LIN {X 0,Y 170.6,Z 451.582,A -85,B 0,C 180,E1 -23444.324,E2 -23444.324} C_VEL
LIN {X 0,Y 174.957,Z 460.923,A -85,B 0,C 180,E1 -23446.93,E2 -23446.93} C_VEL
LIN {X 0,Y 177.388,Z 468.584,A -85,B 0,C 180,E1 -23448.831,E2 -23448.831} C_VEL
LIN {X 0,Y 179.037,Z 479.708,A -85,B 0,C 180,E1 -23451.349,E2 -23451.349} C_VEL
LIN {X 0,Y 179.549,Z 490.973,A -85,B 0,C 180,E1 -23454.045,E2 -23454.045} C_VEL
LIN {X 0,Y 179.158,Z 500.868,A -85,B 0,C 180,E1 -23456.688,E2 -23456.688} C_VEL
LIN {X 0,Y 178.388,Z 507.125,A -85,B 0,C 180,E1 -23458.532,E2 -23458.532} C_VEL
LIN {X 0,Y 174.98,Z 515.955,A -85,B 0,C 180,E1 -23461.185,E2 -23461.185} C_VEL
LIN {X 0,Y 171.784,Z 523.786,A -85,B 0,C 180,E1 -23464.166,E2 -23464.166} C_VEL
LIN {X 0,Y 168.834,Z 530.43,A -85,B 0,C 180,E1 -23467.353,E2 -23467.353} C_VEL
LIN {X 0,Y 166.629,Z 535.281,A -85,B 0,C 180,E1 -23470.28,E2 -23470.28} C_VEL
LIN {X 0,Y 164.441,Z 539.995,A -85,B 0,C 180,E1 -23473.871,E2 -23473.871} C_VEL
LIN {X 0,Y 163.057,Z 543.606,A -85,B 0,C 180,E1 -23477.554,E2 -23477.554} C_VEL
LIN {X 0,Y 162.405,Z 545.468,A -85,B 0,C 180,E1 -23480.032,E2 -23480.032} C_VEL
LIN {X 0,Y 162,Z 546.866,A -85,B 0,C 180,E1 -23482.522,E2 -23482.522} C_VEL
LIN {X 0,Y 161.792,Z 547.866,A -85,B 0,C 180,E1 -23485.016,E2 -23485.016} C_VEL
LIN {X 0,Y 161.766,Z 548.53,A -85,B 0,C 180,E1 -23487.776,E2 -23487.776} C_VEL
LIN {X 0,Y 161.899,Z 548.694,A -85,B 0,C 180,E1 -23490,E2 -23490} C_VEL
LIN {X 0,Y 161.765,Z 548.464,A -85,B 0,C 180,E1 -23492.49,E2 -23492.49} C_VEL
LIN {X 0,Y 161.792,Z 547.845,A -85,B 0,C 180,E1 -23494.984,E2 -23494.984} C_VEL
LIN {X 0,Y 162,Z 546.836,A -85,B 0,C 180,E1 -23497.478,E2 -23497.478} C_VEL
LIN {X 0,Y 162.405,Z 545.424,A -85,B 0,C 180,E1 -23499.968,E2 -23499.968} C_VEL
LIN {X 0,Y 163.457,Z 542.468,A -85,B 0,C 180,E1 -23503.679,E2 -23503.679} C_VEL
LIN {X 0,Y 165.07,Z 538.474,A -85,B 0,C 180,E1 -23507.339,E2 -23507.339} C_VEL
LIN {X 0,Y 167.886,Z 532.345,A -85,B 0,C 180,E1 -23511.487,E2 -23511.487} C_VEL
LIN {X 0,Y 170.867,Z 525.858,A -85,B 0,C 180,E1 -23514.829,E2 -23514.829} C_VEL
LIN {X 0,Y 173.339,Z 519.858,A -85,B 0,C 180,E1 -23517.348,E2 -23517.348} C_VEL
LIN {X 0,Y 174.23,Z 516.073,A -85,B 0,C 180,E1 -23518.815,E2 -23518.815} C_VEL
LIN {X 0,Y 174.205,Z 512.249,A -85,B 0,C 180,E1 -23520.33,E2 -23520.33} C_VEL
LIN {X 0,Y 173.132,Z 504.415,A -85,B 0,C 180,E1 -23523.344,E2 -23523.344} C_VEL
LIN {X 0,Y 172.989,Z 498.624,A -85,B 0,C 180,E1 -23525.198,E2 -23525.198} C_VEL
LIN {X 0,Y 173.249,Z 489.2,A -85,B 0,C 180,E1 -23527.785,E2 -23527.785} C_VEL
LIN {X 0,Y 172.79,Z 479.133,A -85,B 0,C 180,E1 -23530.303,E2 -23530.303} C_VEL
LIN {X 0,Y 171.463,Z 470.4,A -85,B 0,C 180,E1 -23532.456,E2 -23532.456} C_VEL
LIN {X 0,Y 169.332,Z 463.748,A -85,B 0,C 180,E1 -23534.279,E2 -23534.279} C_VEL
LIN {X 0,Y 165.519,Z 455.347,A -85,B 0,C 180,E1 -23536.863,E2 -23536.863} C_VEL
LIN {X 0,Y 163.537,Z 451.389,A -85,B 0,C 180,E1 -23538.129,E2 -23538.129} C_VEL
LIN {X 0,Y 161.489,Z 447.46,A -85,B 0,C 180,E1 -23539.426,E2 -23539.426} C_VEL
LIN {X 0,Y 160.888,Z 446.45,A -85,B 0,C 180,E1 -23539.781,E2 -23539.781} C_VEL
LIN {X 0,Y 158.813,Z 443.395,A -85,B 0,C 180,E1 -23540.997,E2 -23540.997} C_VEL
LIN {X 0,Y 158.112,Z 441.187,A -85,B 0,C 180,E1 -23541.578,E2 -23541.578} C_VEL
LIN {X 0,Y 157.962,Z 439.682,A -85,B 0,C 180,E1 -23544.662,E2 -23544.662} C_VEL
LIN {X 0,Y 157.752,Z 438.263,A -85,B 0,C 180,E1 -23547.829,E2 -23547.829} C_VEL
LIN {X 0,Y 157.341,Z 436.003,A -85,B 0,C 180,E1 -23553.47,E2 -23553.47} C_VEL
LIN {X 0,Y 157.395,Z 435.881,A -85,B 0,C 180,E1 -23559.667,E2 -23559.667} C_VEL
LIN {X 0,Y 157.48,Z 435.869,A -85,B 0,C 180,E1 -23564.469,E2 -23564.469} C_VEL
LIN {X 0,Y 157.774,Z 435.833,A -85,B 0,C 180,E1 -23569.736,E2 -23569.736} C_VEL
LIN {X 0,Y 157.826,Z 435.824,A -85,B 0,C 180,E1 -23572.323,E2 -23572.323} C_VEL
LIN {X 0,Y 158.261,Z 435.77,A -85,B 0,C 180,E1 -23580,E2 -23580} C_VEL
LIN {X 0,Y 157.826,Z 435.825,A -85,B 0,C 180,E1 -23587.677,E2 -23587.677} C_VEL
LIN {X 0,Y 157.707,Z 435.839,A -85,B 0,C 180,E1 -23591.363,E2 -23591.363} C_VEL
LIN {X 0,Y 157.48,Z 435.868,A -85,B 0,C 180,E1 -23595.532,E2 -23595.532} C_VEL
LIN {X 0,Y 157.371,Z 435.88,A -85,B 0,C 180,E1 -23600.933,E2 -23600.933} C_VEL
LIN {X 0,Y 157.316,Z 435.888,A -85,B 0,C 180,E1 -23606.685,E2 -23606.685} C_VEL
LIN {X 0,Y 157.279,Z 435.892,A -85,B 0,C 180,E1 -23612.427,E2 -23612.427} C_VEL
LIN {X 0,Y 157.257,Z 435.896,A -85,B 0,C 180,E1 -23617.476,E2 -23617.476} C_VEL
LIN {X 0,Y 157.227,Z 435.906,A -85,B 0,C 180,E1 -23618.11,E2 -23618.11} C_VEL
LIN {X 0,Y 158.173,Z 438.66,A -85,B 0,C 180,E1 -23618.871,E2 -23618.871} C_VEL
LIN {X 0,Y 160.688,Z 441.686,A -85,B 0,C 180,E1 -23620.309,E2 -23620.309} C_VEL
LIN {X 0,Y 162.705,Z 445.357,A -85,B 0,C 180,E1 -23621.615,E2 -23621.615} C_VEL
LIN {X 0,Y 163.922,Z 447.482,A -85,B 0,C 180,E1 -23622.371,E2 -23622.371} C_VEL
LIN {X 0,Y 166.788,Z 452.918,A -85,B 0,C 180,E1 -23624.248,E2 -23624.248} C_VEL
LIN {X 0,Y 170.183,Z 460.491,A -85,B 0,C 180,E1 -23626.703,E2 -23626.703} C_VEL
LIN {X 0,Y 173.03,Z 469.987,A -85,B 0,C 180,E1 -23629.468,E2 -23629.468} C_VEL
LIN {X 0,Y 174.705,Z 480.999,A -85,B 0,C 180,E1 -23632.557,E2 -23632.557} C_VEL
LIN {X 0,Y 175.044,Z 489.187,A -85,B 0,C 180,E1 -23634.944,E2 -23634.944} C_VEL
LIN {X 0,Y 174.851,Z 495.164,A -85,B 0,C 180,E1 -23636.794,E2 -23636.794} C_VEL
LIN {X 0,Y 171.108,Z 504.928,A -85,B 0,C 180,E1 -23639.604,E2 -23639.604} C_VEL
LIN {X 0,Y 167.634,Z 512.925,A -85,B 0,C 180,E1 -23642.537,E2 -23642.537} C_VEL
LIN {X 0,Y 164.104,Z 520.326,A -85,B 0,C 180,E1 -23645.993,E2 -23645.993} C_VEL
LIN {X 0,Y 161.079,Z 526.265,A -85,B 0,C 180,E1 -23649.571,E2 -23649.571} C_VEL
LIN {X 0,Y 158.726,Z 530.952,A -85,B 0,C 180,E1 -23653.274,E2 -23653.274} C_VEL
LIN {X 0,Y 156.932,Z 534.537,A -85,B 0,C 180,E1 -23657.061,E2 -23657.061} C_VEL
LIN {X 0,Y 156.086,Z 536.386,A -85,B 0,C 180,E1 -23659.624,E2 -23659.624} C_VEL
LIN {X 0,Y 155.506,Z 537.773,A -85,B 0,C 180,E1 -23662.208,E2 -23662.208} C_VEL
LIN {X 0,Y 154.905,Z 539.364,A -85,B 0,C 180,E1 -23667.4,E2 -23667.4} C_VEL
LIN {X 0,Y 154.861,Z 539.59,A -85,B 0,C 180,E1 -23670,E2 -23670} C_VEL
LIN {X 0,Y 155.016,Z 539.119,A -85,B 0,C 180,E1 -23674.11,E2 -23674.11} C_VEL
LIN {X 0,Y 155.506,Z 537.842,A -85,B 0,C 180,E1 -23677.793,E2 -23677.793} C_VEL
LIN {X 0,Y 156.086,Z 536.486,A -85,B 0,C 180,E1 -23680.376,E2 -23680.376} C_VEL
LIN {X 0,Y 157.445,Z 533.617,A -85,B 0,C 180,E1 -23684.212,E2 -23684.212} C_VEL
LIN {X 0,Y 159.414,Z 529.724,A -85,B 0,C 180,E1 -23687.976,E2 -23687.976} C_VEL
LIN {X 0,Y 161.939,Z 524.7,A -85,B 0,C 180,E1 -23691.648,E2 -23691.648} C_VEL
LIN {X 0,Y 165.158,Z 518.366,A -85,B 0,C 180,E1 -23695.185,E2 -23695.185} C_VEL
LIN {X 0,Y 168.668,Z 510.778,A -85,B 0,C 180,E1 -23698.48,E2 -23698.48} C_VEL
LIN {X 0,Y 172.046,Z 502.551,A -85,B 0,C 180,E1 -23701.32,E2 -23701.32} C_VEL
LIN {X 0,Y 175.038,Z 494.65,A -85,B 0,C 180,E1 -23703.51,E2 -23703.51} C_VEL
LIN {X 0,Y 175.053,Z 485.144,A -85,B 0,C 180,E1 -23706.412,E2 -23706.412} C_VEL
LIN {X 0,Y 174.124,Z 476.029,A -85,B 0,C 180,E1 -23709.032,E2 -23709.032} C_VEL
LIN {X 0,Y 172.706,Z 468.444,A -85,B 0,C 180,E1 -23711.162,E2 -23711.162} C_VEL
LIN {X 0,Y 170.166,Z 460.375,A -85,B 0,C 180,E1 -23713.527,E2 -23713.527} C_VEL
LIN {X 0,Y 165.678,Z 450.421,A -85,B 0,C 180,E1 -23716.743,E2 -23716.743} C_VEL
LIN {X 0,Y 163.427,Z 446.317,A -85,B 0,C 180,E1 -23718.197,E2 -23718.197} C_VEL
LIN {X 0,Y 160.984,Z 442.422,A -85,B 0,C 180,E1 -23719.707,E2 -23719.707} C_VEL
LIN {X 0,Y 160.22,Z 440.995,A -85,B 0,C 180,E1 -23720.199,E2 -23720.199} C_VEL
LIN {X 0,Y 157.993,Z 438.397,A -85,B 0,C 180,E1 -23721.481,E2 -23721.481} C_VEL
LIN {X 0,Y 157.227,Z 435.899,A -85,B 0,C 180,E1 -23722.204,E2 -23722.204} C_VEL
LIN {X 0,Y 157.292,Z 435.889,A -85,B 0,C 180,E1 -23724.489,E2 -23724.489} C_VEL
LIN {X 0,Y 157.296,Z 435.89,A -85,B 0,C 180,E1 -23728.095,E2 -23728.095} C_VEL
LIN {X 0,Y 157.324,Z 435.883,A -85,B 0,C 180,E1 -23733.466,E2 -23733.466} C_VEL
LIN {X 0,Y 157.396,Z 435.878,A -85,B 0,C 180,E1 -23739.667,E2 -23739.667} C_VEL
LIN {X 0,Y 157.481,Z 435.868,A -85,B 0,C 180,E1 -23744.468,E2 -23744.468} C_VEL
LIN {X 0,Y 157.775,Z 435.833,A -85,B 0,C 180,E1 -23749.736,E2 -23749.736} C_VEL
LIN {X 0,Y 157.827,Z 435.826,A -85,B 0,C 180,E1 -23752.323,E2 -23752.323} C_VEL
LIN {X 0,Y 158.261,Z 435.77,A -85,B 0,C 180,E1 -23760,E2 -23760} C_VEL
LIN {X 0,Y 157.827,Z 435.824,A -85,B 0,C 180,E1 -23767.677,E2 -23767.677} C_VEL
LIN {X 0,Y 157.708,Z 435.839,A -85,B 0,C 180,E1 -23771.363,E2 -23771.363} C_VEL
LIN {X 0,Y 157.488,Z 435.866,A -85,B 0,C 180,E1 -23775.531,E2 -23775.531} C_VEL
LIN {X 0,Y 157.373,Z 435.882,A -85,B 0,C 180,E1 -23780.932,E2 -23780.932} C_VEL
LIN {X 0,Y 157.382,Z 436.144,A -85,B 0,C 180,E1 -23786.732,E2 -23786.732} C_VEL
LIN {X 0,Y 157.715,Z 438.408,A -85,B 0,C 180,E1 -23792.326,E2 -23792.326} C_VEL
LIN {X 0,Y 158.04,Z 440.801,A -85,B 0,C 180,E1 -23797.515,E2 -23797.515} C_VEL
LIN {X 0,Y 158.138,Z 441.341,A -85,B 0,C 180,E1 -23798.352,E2 -23798.352} C_VEL
LIN {X 0,Y 159.193,Z 444.167,A -85,B 0,C 180,E1 -23799.109,E2 -23799.109} C_VEL
LIN {X 0,Y 161.514,Z 447.463,A -85,B 0,C 180,E1 -23800.447,E2 -23800.447} C_VEL
LIN {X 0,Y 163.398,Z 451.165,A -85,B 0,C 180,E1 -23801.659,E2 -23801.659} C_VEL
LIN {X 0,Y 164.568,Z 453.304,A -85,B 0,C 180,E1 -23802.373,E2 -23802.373} C_VEL
LIN {X 0,Y 168.071,Z 460.658,A -85,B 0,C 180,E1 -23804.694,E2 -23804.694} C_VEL
LIN {X 0,Y 171.256,Z 469.263,A -85,B 0,C 180,E1 -23807.171,E2 -23807.171} C_VEL
LIN {X 0,Y 172.513,Z 476.304,A -85,B 0,C 180,E1 -23808.911,E2 -23808.911} C_VEL
LIN {X 0,Y 173.303,Z 485.676,A -85,B 0,C 180,E1 -23811.238,E2 -23811.238} C_VEL
LIN {X 0,Y 173.202,Z 496.91,A -85,B 0,C 180,E1 -23814.247,E2 -23814.247} C_VEL
LIN {X 0,Y 172.404,Z 504.943,A -85,B 0,C 180,E1 -23816.61,E2 -23816.61} C_VEL
LIN {X 0,Y 171.672,Z 508.87,A -85,B 0,C 180,E1 -23817.845,E2 -23817.845} C_VEL
LIN {X 0,Y 168.103,Z 517.33,A -85,B 0,C 180,E1 -23820.577,E2 -23820.577} C_VEL
LIN {X 0,Y 164.638,Z 525.326,A -85,B 0,C 180,E1 -23823.901,E2 -23823.901} C_VEL
LIN {X 0,Y 161.257,Z 532.261,A -85,B 0,C 180,E1 -23827.582,E2 -23827.582} C_VEL
LIN {X 0,Y 158.296,Z 538.357,A -85,B 0,C 180,E1 -23831.893,E2 -23831.893} C_VEL
LIN {X 0,Y 156.531,Z 542.326,A -85,B 0,C 180,E1 -23835.703,E2 -23835.703} C_VEL
LIN {X 0,Y 155.406,Z 545.264,A -85,B 0,C 180,E1 -23839.578,E2 -23839.578} C_VEL
LIN {X 0,Y 154.95,Z 546.662,A -85,B 0,C 180,E1 -23842.179,E2 -23842.179} C_VEL
LIN {X 0,Y 154.712,Z 547.662,A -85,B 0,C 180,E1 -23844.787,E2 -23844.787} C_VEL
LIN {X 0,Y 154.684,Z 548.389,A -85,B 0,C 180,E1 -23848.304,E2 -23848.304} C_VEL
LIN {X 0,Y 154.797,Z 548.49,A -85,B 0,C 180,E1 -23850,E2 -23850} C_VEL
LIN {X 0,Y 154.667,Z 548.26,A -85,B 0,C 180,E1 -23852.604,E2 -23852.604} C_VEL
LIN {X 0,Y 154.712,Z 547.64,A -85,B 0,C 180,E1 -23855.212,E2 -23855.212} C_VEL
LIN {X 0,Y 154.95,Z 546.631,A -85,B 0,C 180,E1 -23857.82,E2 -23857.82} C_VEL
LIN {X 0,Y 155.405,Z 545.219,A -85,B 0,C 180,E1 -23860.422,E2 -23860.422} C_VEL
LIN {X 0,Y 156.53,Z 542.262,A -85,B 0,C 180,E1 -23864.296,E2 -23864.296} C_VEL
LIN {X 0,Y 158.295,Z 538.269,A -85,B 0,C 180,E1 -23868.106,E2 -23868.106} C_VEL
LIN {X 0,Y 161.255,Z 532.138,A -85,B 0,C 180,E1 -23872.417,E2 -23872.417} C_VEL
LIN {X 0,Y 164.561,Z 525.263,A -85,B 0,C 180,E1 -23876.062,E2 -23876.062} C_VEL
LIN {X 0,Y 168.101,Z 517.147,A -85,B 0,C 180,E1 -23879.422,E2 -23879.422} C_VEL
LIN {X 0,Y 171.631,Z 508.636,A -85,B 0,C 180,E1 -23882.163,E2 -23882.163} C_VEL
LIN {X 0,Y 172.869,Z 500.383,A -85,B 0,C 180,E1 -23884.692,E2 -23884.692} C_VEL
LIN {X 0,Y 172.989,Z 498.624,A -85,B 0,C 180,E1 -23885.198,E2 -23885.198} C_VEL
LIN {X 0,Y 172.681,Z 494.345,A -85,B 0,C 180,E1 -23886.531,E2 -23886.531} C_VEL
LIN {X 0,Y 171.427,Z 490.35,A -85,B 0,C 180,E1 -23887.944,E2 -23887.944} C_VEL
LIN {X 0,Y 168.002,Z 482.617,A -85,B 0,C 180,E1 -23890.835,E2 -23890.835} C_VEL
LIN {X 0,Y 166.494,Z 476.796,A -85,B 0,C 180,E1 -23892.645,E2 -23892.645} C_VEL
LIN {X 0,Y 165.046,Z 470.124,A -85,B 0,C 180,E1 -23894.532,E2 -23894.532} C_VEL
LIN {X 0,Y 161.383,Z 460.851,A -85,B 0,C 180,E1 -23897.547,E2 -23897.547} C_VEL
LIN {X 0,Y 159.089,Z 456.083,A -85,B 0,C 180,E1 -23899.233,E2 -23899.233} C_VEL
LIN {X 0,Y 156.754,Z 451.512,A -85,B 0,C 180,E1 -23900.914,E2 -23900.914} C_VEL
LIN {X 0,Y 154.664,Z 447.676,A -85,B 0,C 180,E1 -23902.409,E2 -23902.409} C_VEL
LIN {X 0,Y 153.912,Z 446.339,A -85,B 0,C 180,E1 -23902.93,E2 -23902.93} C_VEL
LIN {X 0,Y 151.726,Z 443.154,A -85,B 0,C 180,E1 -23904.416,E2 -23904.416} C_VEL
LIN {X 0,Y 150.944,Z 440.831,A -85,B 0,C 180,E1 -23905.224,E2 -23905.224} C_VEL
LIN {X 0,Y 150.666,Z 439.2,A -85,B 0,C 180,E1 -23909.129,E2 -23909.129} C_VEL
LIN {X 0,Y 150.431,Z 437.884,A -85,B 0,C 180,E1 -23912.581,E2 -23912.581} C_VEL
LIN {X 0,Y 150.266,Z 436.997,A -85,B 0,C 180,E1 -23915.106,E2 -23915.106} C_VEL
LIN {X 0,Y 150.368,Z 436.756,A -85,B 0,C 180,E1 -23920.903,E2 -23920.903} C_VEL
LIN {X 0,Y 150.465,Z 436.742,A -85,B 0,C 180,E1 -23926.494,E2 -23926.494} C_VEL
LIN {X 0,Y 150.69,Z 436.715,A -85,B 0,C 180,E1 -23929.248,E2 -23929.248} C_VEL
LIN {X 0,Y 150.764,Z 436.706,A -85,B 0,C 180,E1 -23931.961,E2 -23931.961} C_VEL
LIN {X 0,Y 151.221,Z 436.647,A -85,B 0,C 180,E1 -23940,E2 -23940} C_VEL
LIN {X 0,Y 150.764,Z 436.704,A -85,B 0,C 180,E1 -23948.039,E2 -23948.039} C_VEL
LIN {X 0,Y 150.636,Z 436.72,A -85,B 0,C 180,E1 -23951.546,E2 -23951.546} C_VEL
LIN {X 0,Y 150.385,Z 436.751,A -85,B 0,C 180,E1 -23956.284,E2 -23956.284} C_VEL
LIN {X 0,Y 150.352,Z 436.753,A -85,B 0,C 180,E1 -23960.793,E2 -23960.793} C_VEL
LIN {X 0,Y 150.245,Z 436.768,A -85,B 0,C 180,E1 -23967.283,E2 -23967.283} C_VEL
LIN {X 0,Y 150.22,Z 436.771,A -85,B 0,C 180,E1 -23972.635,E2 -23972.635} C_VEL
LIN {X 0,Y 150.222,Z 436.885,A -85,B 0,C 180,E1 -23974.661,E2 -23974.661} C_VEL
LIN {X 0,Y 151.09,Z 439.359,A -85,B 0,C 180,E1 -23975.45,E2 -23975.45} C_VEL
LIN {X 0,Y 153.214,Z 441.722,A -85,B 0,C 180,E1 -23976.852,E2 -23976.852} C_VEL
LIN {X 0,Y 153.8,Z 442.446,A -85,B 0,C 180,E1 -23977.238,E2 -23977.238} C_VEL
LIN {X 0,Y 155.53,Z 445.479,A -85,B 0,C 180,E1 -23978.515,E2 -23978.515} C_VEL
LIN {X 0,Y 156.95,Z 447.413,A -85,B 0,C 180,E1 -23979.442,E2 -23979.442} C_VEL
LIN {X 0,Y 160.981,Z 455.021,A -85,B 0,C 180,E1 -23982.416,E2 -23982.416} C_VEL
LIN {X 0,Y 164.913,Z 464.218,A -85,B 0,C 180,E1 -23985.651,E2 -23985.651} C_VEL
LIN {X 0,Y 167.208,Z 472.415,A -85,B 0,C 180,E1 -23988.25,E2 -23988.25} C_VEL
LIN {X 0,Y 168.59,Z 482.499,A -85,B 0,C 180,E1 -23991.296,E2 -23991.296} C_VEL
LIN {X 0,Y 168.823,Z 491.095,A -85,B 0,C 180,E1 -23993.988,E2 -23993.988} C_VEL
LIN {X 0,Y 168.559,Z 496.426,A -85,B 0,C 180,E1 -23995.745,E2 -23995.745} C_VEL
LIN {X 0,Y 164.739,Z 505.744,A -85,B 0,C 180,E1 -23998.565,E2 -23998.565} C_VEL
LIN {X 0,Y 160.736,Z 514.478,A -85,B 0,C 180,E1 -24001.964,E2 -24001.964} C_VEL
LIN {X 0,Y 157.062,Z 521.642,A -85,B 0,C 180,E1 -24005.55,E2 -24005.55} C_VEL
LIN {X 0,Y 154.431,Z 526.471,A -85,B 0,C 180,E1 -24008.65,E2 -24008.65} C_VEL
LIN {X 0,Y 151.949,Z 531.157,A -85,B 0,C 180,E1 -24012.504,E2 -24012.504} C_VEL
LIN {X 0,Y 150.017,Z 534.742,A -85,B 0,C 180,E1 -24016.453,E2 -24016.453} C_VEL
LIN {X 0,Y 149.111,Z 536.591,A -85,B 0,C 180,E1 -24019.133,E2 -24019.133} C_VEL
LIN {X 0,Y 148.469,Z 537.977,A -85,B 0,C 180,E1 -24021.836,E2 -24021.836} C_VEL
LIN {X 0,Y 147.854,Z 539.446,A -85,B 0,C 180,E1 -24026.567,E2 -24026.567} C_VEL
LIN {X 0,Y 147.766,Z 539.794,A -85,B 0,C 180,E1 -24030,E2 -24030} C_VEL
LIN {X 0,Y 147.854,Z 539.476,A -85,B 0,C 180,E1 -24033.431,E2 -24033.431} C_VEL
LIN {X 0,Y 148.469,Z 538.046,A -85,B 0,C 180,E1 -24038.164,E2 -24038.164} C_VEL
LIN {X 0,Y 149.111,Z 536.689,A -85,B 0,C 180,E1 -24040.867,E2 -24040.867} C_VEL
LIN {X 0,Y 150.573,Z 533.82,A -85,B 0,C 180,E1 -24044.875,E2 -24044.875} C_VEL
LIN {X 0,Y 152.685,Z 529.926,A -85,B 0,C 180,E1 -24048.797,E2 -24048.797} C_VEL
LIN {X 0,Y 155.372,Z 524.903,A -85,B 0,C 180,E1 -24052.612,E2 -24052.612} C_VEL
LIN {X 0,Y 158.768,Z 518.568,A -85,B 0,C 180,E1 -24056.274,E2 -24056.274} C_VEL
LIN {X 0,Y 162.327,Z 511.235,A -85,B 0,C 180,E1 -24059.578,E2 -24059.578} C_VEL
LIN {X 0,Y 166.011,Z 502.753,A -85,B 0,C 180,E1 -24062.596,E2 -24062.596} C_VEL
LIN {X 0,Y 168.729,Z 495.917,A -85,B 0,C 180,E1 -24064.578,E2 -24064.578} C_VEL
LIN {X 0,Y 168.945,Z 487.996,A -85,B 0,C 180,E1 -24067.165,E2 -24067.165} C_VEL
LIN {X 0,Y 168.274,Z 478.859,A -85,B 0,C 180,E1 -24069.991,E2 -24069.991} C_VEL
LIN {X 0,Y 166.957,Z 471.09,A -85,B 0,C 180,E1 -24072.339,E2 -24072.339} C_VEL
LIN {X 0,Y 164.899,Z 464.066,A -85,B 0,C 180,E1 -24074.599,E2 -24074.599} C_VEL
LIN {X 0,Y 161.209,Z 455.356,A -85,B 0,C 180,E1 -24077.658,E2 -24077.658} C_VEL
LIN {X 0,Y 158.247,Z 449.966,A -85,B 0,C 180,E1 -24079.807,E2 -24079.807} C_VEL
LIN {X 0,Y 156.422,Z 446.511,A -85,B 0,C 180,E1 -24081.167,E2 -24081.167} C_VEL
LIN {X 0,Y 154.251,Z 443.523,A -85,B 0,C 180,E1 -24082.634,E2 -24082.634} C_VEL
LIN {X 0,Y 153.512,Z 441.903,A -85,B 0,C 180,E1 -24083.232,E2 -24083.232} C_VEL
LIN {X 0,Y 151.255,Z 439.601,A -85,B 0,C 180,E1 -24084.696,E2 -24084.696} C_VEL
LIN {X 0,Y 150.266,Z 437.159,A -85,B 0,C 180,E1 -24085.554,E2 -24085.554} C_VEL
LIN {X 0,Y 150.189,Z 436.777,A -85,B 0,C 180,E1 -24085.737,E2 -24085.737} C_VEL
LIN {X 0,Y 150.209,Z 436.774,A -85,B 0,C 180,E1 -24089.024,E2 -24089.024} C_VEL
LIN {X 0,Y 150.246,Z 436.769,A -85,B 0,C 180,E1 -24092.718,E2 -24092.718} C_VEL
LIN {X 0,Y 150.353,Z 436.756,A -85,B 0,C 180,E1 -24099.207,E2 -24099.207} C_VEL
LIN {X 0,Y 150.385,Z 436.753,A -85,B 0,C 180,E1 -24103.716,E2 -24103.716} C_VEL
LIN {X 0,Y 150.692,Z 436.714,A -85,B 0,C 180,E1 -24109.248,E2 -24109.248} C_VEL
LIN {X 0,Y 150.766,Z 436.704,A -85,B 0,C 180,E1 -24111.961,E2 -24111.961} C_VEL
LIN {X 0,Y 151.221,Z 436.646,A -85,B 0,C 180,E1 -24120,E2 -24120} C_VEL
LIN {X 0,Y 150.766,Z 436.703,A -85,B 0,C 180,E1 -24128.039,E2 -24128.039} C_VEL
LIN {X 0,Y 150.637,Z 436.72,A -85,B 0,C 180,E1 -24131.546,E2 -24131.546} C_VEL
LIN {X 0,Y 150.393,Z 436.751,A -85,B 0,C 180,E1 -24136.283,E2 -24136.283} C_VEL
LIN {X 0,Y 150.354,Z 436.756,A -85,B 0,C 180,E1 -24140.794,E2 -24140.794} C_VEL
LIN {X 0,Y 150.31,Z 437.057,A -85,B 0,C 180,E1 -24144.886,E2 -24144.886} C_VEL
LIN {X 0,Y 150.491,Z 438.102,A -85,B 0,C 180,E1 -24147.84,E2 -24147.84} C_VEL
LIN {X 0,Y 150.78,Z 440.132,A -85,B 0,C 180,E1 -24152.965,E2 -24152.965} C_VEL
LIN {X 0,Y 150.906,Z 440.865,A -85,B 0,C 180,E1 -24154.684,E2 -24154.684} C_VEL
LIN {X 0,Y 152.284,Z 444.264,A -85,B 0,C 180,E1 -24155.841,E2 -24155.841} C_VEL
LIN {X 0,Y 154.422,Z 447.057,A -85,B 0,C 180,E1 -24157.242,E2 -24157.242} C_VEL
LIN {X 0,Y 156.347,Z 450.939,A -85,B 0,C 180,E1 -24158.675,E2 -24158.675} C_VEL
LIN {X 0,Y 157.545,Z 452.854,A -85,B 0,C 180,E1 -24159.471,E2 -24159.471} C_VEL
LIN {X 0,Y 160.381,Z 458.671,A -85,B 0,C 180,E1 -24161.554,E2 -24161.554} C_VEL
LIN {X 0,Y 164.156,Z 467.609,A -85,B 0,C 180,E1 -24164.565,E2 -24164.565} C_VEL
LIN {X 0,Y 166.074,Z 473.749,A -85,B 0,C 180,E1 -24166.447,E2 -24166.447} C_VEL
LIN {X 0,Y 167.183,Z 484.005,A -85,B 0,C 180,E1 -24169.173,E2 -24169.173} C_VEL
LIN {X 0,Y 167.163,Z 494.392,A -85,B 0,C 180,E1 -24172.032,E2 -24172.032} C_VEL
LIN {X 0,Y 166.384,Z 503.689,A -85,B 0,C 180,E1 -24174.864,E2 -24174.864} C_VEL
LIN {X 0,Y 165.529,Z 508.663,A -85,B 0,C 180,E1 -24176.499,E2 -24176.499} C_VEL
LIN {X 0,Y 161.933,Z 517.128,A -85,B 0,C 180,E1 -24179.339,E2 -24179.339} C_VEL
LIN {X 0,Y 158.439,Z 524.637,A -85,B 0,C 180,E1 -24182.518,E2 -24182.518} C_VEL
LIN {X 0,Y 155.237,Z 531.045,A -85,B 0,C 180,E1 -24185.955,E2 -24185.955} C_VEL
LIN {X 0,Y 152.373,Z 536.565,A -85,B 0,C 180,E1 -24189.761,E2 -24189.761} C_VEL
LIN {X 0,Y 150.14,Z 540.897,A -85,B 0,C 180,E1 -24193.688,E2 -24193.688} C_VEL
LIN {X 0,Y 149.141,Z 543.197,A -85,B 0,C 180,E1 -24196.372,E2 -24196.372} C_VEL
LIN {X 0,Y 148.392,Z 545.059,A -85,B 0,C 180,E1 -24199.079,E2 -24199.079} C_VEL
LIN {X 0,Y 147.899,Z 546.458,A -85,B 0,C 180,E1 -24201.804,E2 -24201.804} C_VEL
LIN {X 0,Y 147.635,Z 547.458,A -85,B 0,C 180,E1 -24204.536,E2 -24204.536} C_VEL
LIN {X 0,Y 147.622,Z 548.22,A -85,B 0,C 180,E1 -24208.772,E2 -24208.772} C_VEL
LIN {X 0,Y 147.63,Z 548.207,A -85,B 0,C 180,E1 -24211.362,E2 -24211.362} C_VEL
LIN {X 0,Y 147.634,Z 547.436,A -85,B 0,C 180,E1 -24215.463,E2 -24215.463} C_VEL
LIN {X 0,Y 147.899,Z 546.426,A -85,B 0,C 180,E1 -24218.196,E2 -24218.196} C_VEL
LIN {X 0,Y 148.392,Z 545.013,A -85,B 0,C 180,E1 -24220.92,E2 -24220.92} C_VEL
LIN {X 0,Y 149.629,Z 542.057,A -85,B 0,C 180,E1 -24224.971,E2 -24224.971} C_VEL
LIN {X 0,Y 151.551,Z 538.063,A -85,B 0,C 180,E1 -24228.942,E2 -24228.942} C_VEL
LIN {X 0,Y 154.687,Z 531.931,A -85,B 0,C 180,E1 -24233.425,E2 -24233.425} C_VEL
LIN {X 0,Y 157.863,Z 525.699,A -85,B 0,C 180,E1 -24236.885,E2 -24236.885} C_VEL
LIN {X 0,Y 161.931,Z 516.94,A -85,B 0,C 180,E1 -24240.661,E2 -24240.661} C_VEL
LIN {X 0,Y 164.883,Z 510.235,A -85,B 0,C 180,E1 -24242.919,E2 -24242.919} C_VEL
LIN {X 0,Y 166.191,Z 504.476,A -85,B 0,C 180,E1 -24244.813,E2 -24244.813} C_VEL
LIN {X 0,Y 167.018,Z 495.396,A -85,B 0,C 180,E1 -24247.609,E2 -24247.609} C_VEL
LIN {X 0,Y 167.155,Z 484.687,A -85,B 0,C 180,E1 -24250.563,E2 -24250.563} C_VEL
LIN {X 0,Y 166.494,Z 476.796,A -85,B 0,C 180,E1 -24252.645,E2 -24252.645} C_VEL
LIN {X 0,Y 165.745,Z 473.947,A -85,B 0,C 180,E1 -24253.532,E2 -24253.532} C_VEL
LIN {X 0,Y 163.6,Z 470.472,A -85,B 0,C 180,E1 -24255.022,E2 -24255.022} C_VEL
LIN {X 0,Y 156.015,Z 462.883,A -85,B 0,C 180,E1 -24259.38,E2 -24259.38} C_VEL
LIN {X 0,Y 153.866,Z 459.161,A -85,B 0,C 180,E1 -24260.966,E2 -24260.966} C_VEL
LIN {X 0,Y 152.646,Z 456.604,A -85,B 0,C 180,E1 -24261.98,E2 -24261.98} C_VEL
LIN {X 0,Y 150.11,Z 451.657,A -85,B 0,C 180,E1 -24264.077,E2 -24264.077} C_VEL
LIN {X 0,Y 147.958,Z 447.937,A -85,B 0,C 180,E1 -24265.83,E2 -24265.83} C_VEL
LIN {X 0,Y 147.298,Z 446.533,A -85,B 0,C 180,E1 -24266.41,E2 -24266.41} C_VEL
LIN {X 0,Y 144.714,Z 443.295,A -85,B 0,C 180,E1 -24268.427,E2 -24268.427} C_VEL
LIN {X 0,Y 143.691,Z 440.536,A -85,B 0,C 180,E1 -24269.506,E2 -24269.506} C_VEL
LIN {X 0,Y 143.386,Z 439.002,A -85,B 0,C 180,E1 -24273.824,E2 -24273.824} C_VEL
LIN {X 0,Y 143.278,Z 437.638,A -85,B 0,C 180,E1 -24278.745,E2 -24278.745} C_VEL
LIN {X 0,Y 143.318,Z 437.634,A -85,B 0,C 180,E1 -24282.889,E2 -24282.889} C_VEL
LIN {X 0,Y 143.604,Z 437.597,A -85,B 0,C 180,E1 -24288.711,E2 -24288.711} C_VEL
LIN {X 0,Y 143.686,Z 437.587,A -85,B 0,C 180,E1 -24291.562,E2 -24291.562} C_VEL
LIN {X 0,Y 144.18,Z 437.524,A -85,B 0,C 180,E1 -24300,E2 -24300} C_VEL
LIN {X 0,Y 143.686,Z 437.585,A -85,B 0,C 180,E1 -24308.438,E2 -24308.438} C_VEL
LIN {X 0,Y 143.572,Z 437.601,A -85,B 0,C 180,E1 -24311.758,E2 -24311.758} C_VEL
LIN {X 0,Y 143.318,Z 437.633,A -85,B 0,C 180,E1 -24317.111,E2 -24317.111} C_VEL
LIN {X 0,Y 143.278,Z 437.637,A -85,B 0,C 180,E1 -24321.255,E2 -24321.255} C_VEL
LIN {X 0,Y 143.192,Z 437.649,A -85,B 0,C 180,E1 -24327.938,E2 -24327.938} C_VEL
LIN {X 0,Y 143.162,Z 437.856,A -85,B 0,C 180,E1 -24330.415,E2 -24330.415} C_VEL
LIN {X 0,Y 144.181,Z 440.493,A -85,B 0,C 180,E1 -24331.499,E2 -24331.499} C_VEL
LIN {X 0,Y 146.135,Z 442.59,A -85,B 0,C 180,E1 -24333.041,E2 -24333.041} C_VEL
LIN {X 0,Y 147.043,Z 443.415,A -85,B 0,C 180,E1 -24333.723,E2 -24333.723} C_VEL
LIN {X 0,Y 148.898,Z 446.679,A -85,B 0,C 180,E1 -24335.325,E2 -24335.325} C_VEL
LIN {X 0,Y 150.328,Z 448.406,A -85,B 0,C 180,E1 -24336.381,E2 -24336.381} C_VEL
LIN {X 0,Y 154.264,Z 455.426,A -85,B 0,C 180,E1 -24339.629,E2 -24339.629} C_VEL
LIN {X 0,Y 158.036,Z 463.592,A -85,B 0,C 180,E1 -24342.945,E2 -24342.945} C_VEL
LIN {X 0,Y 160.425,Z 470.492,A -85,B 0,C 180,E1 -24345.498,E2 -24345.498} C_VEL
LIN {X 0,Y 161.963,Z 478.087,A -85,B 0,C 180,E1 -24348.027,E2 -24348.027} C_VEL
LIN {X 0,Y 162.734,Z 487.182,A -85,B 0,C 180,E1 -24351.021,E2 -24351.021} C_VEL
LIN {X 0,Y 162.478,Z 495.604,A -85,B 0,C 180,E1 -24353.889,E2 -24353.889} C_VEL
LIN {X 0,Y 161.901,Z 498.586,A -85,B 0,C 180,E1 -24354.889,E2 -24354.889} C_VEL
LIN {X 0,Y 157.566,Z 508.467,A -85,B 0,C 180,E1 -24358.134,E2 -24358.134} C_VEL
LIN {X 0,Y 153.838,Z 516.01,A -85,B 0,C 180,E1 -24361.335,E2 -24361.335} C_VEL
LIN {X 0,Y 150.035,Z 522.873,A -85,B 0,C 180,E1 -24365.066,E2 -24365.066} C_VEL
LIN {X 0,Y 146.912,Z 528.363,A -85,B 0,C 180,E1 -24368.975,E2 -24368.975} C_VEL
LIN {X 0,Y 144.424,Z 532.67,A -85,B 0,C 180,E1 -24373.024,E2 -24373.024} C_VEL
LIN {X 0,Y 143.13,Z 534.947,A -85,B 0,C 180,E1 -24375.788,E2 -24375.788} C_VEL
LIN {X 0,Y 142.138,Z 536.796,A -85,B 0,C 180,E1 -24378.593,E2 -24378.593} C_VEL
LIN {X 0,Y 141.434,Z 538.182,A -85,B 0,C 180,E1 -24381.427,E2 -24381.427} C_VEL
LIN {X 0,Y 141.007,Z 539.167,A -85,B 0,C 180,E1 -24384.279,E2 -24384.279} C_VEL
LIN {X 0,Y 140.736,Z 539.772,A -85,B 0,C 180,E1 -24387.138,E2 -24387.138} C_VEL
LIN {X 0,Y 140.69,Z 539.997,A -85,B 0,C 180,E1 -24390,E2 -24390} C_VEL
LIN {X 0,Y 140.737,Z 539.802,A -85,B 0,C 180,E1 -24392.863,E2 -24392.863} C_VEL
LIN {X 0,Y 141.007,Z 539.215,A -85,B 0,C 180,E1 -24395.721,E2 -24395.721} C_VEL
LIN {X 0,Y 142.137,Z 536.893,A -85,B 0,C 180,E1 -24401.408,E2 -24401.408} C_VEL
LIN {X 0,Y 143.731,Z 534.023,A -85,B 0,C 180,E1 -24405.601,E2 -24405.601} C_VEL
LIN {X 0,Y 145.967,Z 530.13,A -85,B 0,C 180,E1 -24409.697,E2 -24409.697} C_VEL
LIN {X 0,Y 148.827,Z 525.106,A -85,B 0,C 180,E1 -24413.666,E2 -24413.666} C_VEL
LIN {X 0,Y 152.444,Z 518.77,A -85,B 0,C 180,E1 -24417.454,E2 -24417.454} C_VEL
LIN {X 0,Y 155.948,Z 511.918,A -85,B 0,C 180,E1 -24420.673,E2 -24420.673} C_VEL
LIN {X 0,Y 160.148,Z 502.777,A -85,B 0,C 180,E1 -24424.024,E2 -24424.024} C_VEL
LIN {X 0,Y 162.46,Z 497.136,A -85,B 0,C 180,E1 -24425.733,E2 -24425.733} C_VEL
LIN {X 0,Y 162.837,Z 489.361,A -85,B 0,C 180,E1 -24428.42,E2 -24428.42} C_VEL
LIN {X 0,Y 162.361,Z 481.188,A -85,B 0,C 180,E1 -24431.143,E2 -24431.143} C_VEL
LIN {X 0,Y 161.287,Z 473.785,A -85,B 0,C 180,E1 -24433.58,E2 -24433.58} C_VEL
LIN {X 0,Y 159.506,Z 467.435,A -85,B 0,C 180,E1 -24435.808,E2 -24435.808} C_VEL
LIN {X 0,Y 156.667,Z 460.218,A -85,B 0,C 180,E1 -24438.572,E2 -24438.572} C_VEL
LIN {X 0,Y 152.344,Z 451.761,A -85,B 0,C 180,E1 -24442.236,E2 -24442.236} C_VEL
LIN {X 0,Y 150.288,Z 448.329,A -85,B 0,C 180,E1 -24443.919,E2 -24443.919} C_VEL
LIN {X 0,Y 147.423,Z 444.318,A -85,B 0,C 180,E1 -24446.182,E2 -24446.182} C_VEL
LIN {X 0,Y 146.761,Z 442.954,A -85,B 0,C 180,E1 -24446.808,E2 -24446.808} C_VEL
LIN {X 0,Y 144.448,Z 440.912,A -85,B 0,C 180,E1 -24448.566,E2 -24448.566} C_VEL
LIN {X 0,Y 143.285,Z 438.487,A -85,B 0,C 180,E1 -24449.716,E2 -24449.716} C_VEL
LIN {X 0,Y 143.122,Z 437.652,A -85,B 0,C 180,E1 -24449.983,E2 -24449.983} C_VEL
LIN {X 0,Y 143.161,Z 437.645,A -85,B 0,C 180,E1 -24453.779,E2 -24453.779} C_VEL
LIN {X 0,Y 143.312,Z 437.632,A -85,B 0,C 180,E1 -24459.923,E2 -24459.923} C_VEL
LIN {X 0,Y 143.383,Z 437.623,A -85,B 0,C 180,E1 -24465.813,E2 -24465.813} C_VEL
LIN {X 0,Y 143.605,Z 437.596,A -85,B 0,C 180,E1 -24468.711,E2 -24468.711} C_VEL
LIN {X 0,Y 143.687,Z 437.584,A -85,B 0,C 180,E1 -24471.562,E2 -24471.562} C_VEL
LIN {X 0,Y 144.18,Z 437.523,A -85,B 0,C 180,E1 -24480,E2 -24480} C_VEL
LIN {X 0,Y 143.687,Z 437.585,A -85,B 0,C 180,E1 -24488.438,E2 -24488.438} C_VEL
LIN {X 0,Y 143.573,Z 437.601,A -85,B 0,C 180,E1 -24491.757,E2 -24491.757} C_VEL
LIN {X 0,Y 143.326,Z 437.632,A -85,B 0,C 180,E1 -24497.11,E2 -24497.11} C_VEL
LIN {X 0,Y 143.28,Z 437.639,A -85,B 0,C 180,E1 -24501.256,E2 -24501.256} C_VEL
LIN {X 0,Y 143.566,Z 439.768,A -85,B 0,C 180,E1 -24508.217,E2 -24508.217} C_VEL
LIN {X 0,Y 143.653,Z 440.569,A -85,B 0,C 180,E1 -24510.3,E2 -24510.3} C_VEL
LIN {X 0,Y 144.889,Z 443.654,A -85,B 0,C 180,E1 -24511.531,E2 -24511.531} C_VEL
LIN {X 0,Y 147.284,Z 446.558,A -85,B 0,C 180,E1 -24513.396,E2 -24513.396} C_VEL
LIN {X 0,Y 149.763,Z 451.228,A -85,B 0,C 180,E1 -24515.502,E2 -24515.502} C_VEL
LIN {X 0,Y 150.946,Z 453.149,A -85,B 0,C 180,E1 -24516.416,E2 -24516.416} C_VEL
LIN {X 0,Y 153.334,Z 457.813,A -85,B 0,C 180,E1 -24518.394,E2 -24518.394} C_VEL
LIN {X 0,Y 156.79,Z 465.544,A -85,B 0,C 180,E1 -24521.388,E2 -24521.388} C_VEL
LIN {X 0,Y 160.046,Z 474.75,A -85,B 0,C 180,E1 -24524.636,E2 -24524.636} C_VEL
LIN {X 0,Y 160.902,Z 479.59,A -85,B 0,C 180,E1 -24526.111,E2 -24526.111} C_VEL
LIN {X 0,Y 161.328,Z 488.098,A -85,B 0,C 180,E1 -24528.558,E2 -24528.558} C_VEL
LIN {X 0,Y 160.794,Z 499.115,A -85,B 0,C 180,E1 -24531.882,E2 -24531.882} C_VEL
LIN {X 0,Y 159.781,Z 506.494,A -85,B 0,C 180,E1 -24534.352,E2 -24534.352} C_VEL
LIN {X 0,Y 158.907,Z 510.258,A -85,B 0,C 180,E1 -24535.674,E2 -24535.674} C_VEL
LIN {X 0,Y 154.395,Z 519.904,A -85,B 0,C 180,E1 -24539.196,E2 -24539.196} C_VEL
LIN {X 0,Y 150.562,Z 527.585,A -85,B 0,C 180,E1 -24542.927,E2 -24542.927} C_VEL
LIN {X 0,Y 146.663,Z 534.67,A -85,B 0,C 180,E1 -24547.458,E2 -24547.458} C_VEL
LIN {X 0,Y 144.029,Z 539.384,A -85,B 0,C 180,E1 -24551.508,E2 -24551.508} C_VEL
LIN {X 0,Y 142.224,Z 542.993,A -85,B 0,C 180,E1 -24555.695,E2 -24555.695} C_VEL
LIN {X 0,Y 141.402,Z 544.855,A -85,B 0,C 180,E1 -24558.532,E2 -24558.532} C_VEL
LIN {X 0,Y 140.85,Z 546.253,A -85,B 0,C 180,E1 -24561.391,E2 -24561.391} C_VEL
LIN {X 0,Y 140.555,Z 547.254,A -85,B 0,C 180,E1 -24564.26,E2 -24564.26} C_VEL
LIN {X 0,Y 140.569,Z 548.054,A -85,B 0,C 180,E1 -24569.356,E2 -24569.356} C_VEL
LIN {X 0,Y 140.487,Z 547.852,A -85,B 0,C 180,E1 -24572.867,E2 -24572.867} C_VEL
LIN {X 0,Y 140.555,Z 547.231,A -85,B 0,C 180,E1 -24575.739,E2 -24575.739} C_VEL
LIN {X 0,Y 140.85,Z 546.221,A -85,B 0,C 180,E1 -24578.609,E2 -24578.609} C_VEL
LIN {X 0,Y 141.402,Z 544.808,A -85,B 0,C 180,E1 -24581.467,E2 -24581.467} C_VEL
LIN {X 0,Y 142.731,Z 541.85,A -85,B 0,C 180,E1 -24585.713,E2 -24585.713} C_VEL
LIN {X 0,Y 144.817,Z 537.857,A -85,B 0,C 180,E1 -24589.859,E2 -24589.859} C_VEL
LIN {X 0,Y 148.182,Z 531.725,A -85,B 0,C 180,E1 -24594.519,E2 -24594.519} C_VEL
LIN {X 0,Y 151.95,Z 524.7,A -85,B 0,C 180,E1 -24598.503,E2 -24598.503} C_VEL
LIN {X 0,Y 155.837,Z 516.732,A -85,B 0,C 180,E1 -24601.999,E2 -24601.999} C_VEL
LIN {X 0,Y 158.863,Z 510.024,A -85,B 0,C 180,E1 -24604.336,E2 -24604.336} C_VEL
LIN {X 0,Y 160.289,Z 502.688,A -85,B 0,C 180,E1 -24606.866,E2 -24606.866} C_VEL
LIN {X 0,Y 161.03,Z 493.914,A -85,B 0,C 180,E1 -24609.663,E2 -24609.663} C_VEL
LIN {X 0,Y 161.22,Z 485.27,A -85,B 0,C 180,E1 -24612.177,E2 -24612.177} C_VEL
LIN {X 0,Y 160.519,Z 477.254,A -85,B 0,C 180,E1 -24614.469,E2 -24614.469} C_VEL
LIN {X 0,Y 158.653,Z 470.541,A -85,B 0,C 180,E1 -24616.695,E2 -24616.695} C_VEL
LIN {X 0,Y 155.252,Z 461.897,A -85,B 0,C 180,E1 -24619.829,E2 -24619.829} C_VEL
LIN {X 0,Y 153.866,Z 459.161,A -85,B 0,C 180,E1 -24620.966,E2 -24620.966} C_VEL
LIN {X 0,Y 152.429,Z 456.91,A -85,B 0,C 180,E1 -24622.036,E2 -24622.036} C_VEL
LIN {X 0,Y 150.519,Z 455.476,A -85,B 0,C 180,E1 -24623.236,E2 -24623.236} C_VEL
LIN {X 0,Y 144.277,Z 452.58,A -85,B 0,C 180,E1 -24627.193,E2 -24627.193} C_VEL
LIN {X 0,Y 143.691,Z 452.07,A -85,B 0,C 180,E1 -24627.642,E2 -24627.642} C_VEL
LIN {X 0,Y 141.391,Z 448.559,A -85,B 0,C 180,E1 -24629.783,E2 -24629.783} C_VEL
LIN {X 0,Y 140.43,Z 446.437,A -85,B 0,C 180,E1 -24630.849,E2 -24630.849} C_VEL
LIN {X 0,Y 137.767,Z 443.49,A -85,B 0,C 180,E1 -24633.387,E2 -24633.387} C_VEL
LIN {X 0,Y 136.432,Z 440.434,A -85,B 0,C 180,E1 -24635.054,E2 -24635.054} C_VEL
LIN {X 0,Y 136.316,Z 439.983,A -85,B 0,C 180,E1 -24635.641,E2 -24635.641} C_VEL
LIN {X 0,Y 136.313,Z 439.014,A -85,B 0,C 180,E1 -24638.844,E2 -24638.844} C_VEL
LIN {X 0,Y 136.253,Z 438.514,A -85,B 0,C 180,E1 -24641.972,E2 -24641.972} C_VEL
LIN {X 0,Y 136.502,Z 438.481,A -85,B 0,C 180,E1 -24648.115,E2 -24648.115} C_VEL
LIN {X 0,Y 136.61,Z 438.468,A -85,B 0,C 180,E1 -24651.122,E2 -24651.122} C_VEL
LIN {X 0,Y 137.137,Z 438.401,A -85,B 0,C 180,E1 -24660,E2 -24660} C_VEL
LIN {X 0,Y 136.61,Z 438.468,A -85,B 0,C 180,E1 -24668.879,E2 -24668.879} C_VEL
LIN {X 0,Y 136.494,Z 438.483,A -85,B 0,C 180,E1 -24671.958,E2 -24671.958} C_VEL
LIN {X 0,Y 136.253,Z 438.509,A -85,B 0,C 180,E1 -24678.028,E2 -24678.028} C_VEL
LIN {X 0,Y 136.199,Z 438.52,A -85,B 0,C 180,E1 -24681.749,E2 -24681.749} C_VEL
LIN {X 0,Y 136.081,Z 438.544,A -85,B 0,C 180,E1 -24684.913,E2 -24684.913} C_VEL
LIN {X 0,Y 136.947,Z 441.092,A -85,B 0,C 180,E1 -24686.17,E2 -24686.17} C_VEL
LIN {X 0,Y 139.006,Z 443.403,A -85,B 0,C 180,E1 -24688.278,E2 -24688.278} C_VEL
LIN {X 0,Y 140.318,Z 444.492,A -85,B 0,C 180,E1 -24689.494,E2 -24689.494} C_VEL
LIN {X 0,Y 141.934,Z 447.514,A -85,B 0,C 180,E1 -24691.223,E2 -24691.223} C_VEL
LIN {X 0,Y 143.782,Z 449.508,A -85,B 0,C 180,E1 -24692.838,E2 -24692.838} C_VEL
LIN {X 0,Y 145.851,Z 452.96,A -85,B 0,C 180,E1 -24694.8,E2 -24694.8} C_VEL
LIN {X 0,Y 148.327,Z 457.112,A -85,B 0,C 180,E1 -24697.081,E2 -24697.081} C_VEL
LIN {X 0,Y 151.711,Z 464.346,A -85,B 0,C 180,E1 -24700.433,E2 -24700.433} C_VEL
LIN {X 0,Y 154.645,Z 472.651,A -85,B 0,C 180,E1 -24703.873,E2 -24703.873} C_VEL
LIN {X 0,Y 156.116,Z 479.866,A -85,B 0,C 180,E1 -24706.545,E2 -24706.545} C_VEL
LIN {X 0,Y 156.717,Z 489.618,A -85,B 0,C 180,E1 -24710.003,E2 -24710.003} C_VEL
LIN {X 0,Y 156.307,Z 496.867,A -85,B 0,C 180,E1 -24712.628,E2 -24712.628} C_VEL
LIN {X 0,Y 156.026,Z 498.798,A -85,B 0,C 180,E1 -24713.357,E2 -24713.357} C_VEL
LIN {X 0,Y 152.072,Z 507.615,A -85,B 0,C 180,E1 -24716.319,E2 -24716.319} C_VEL
LIN {X 0,Y 147.65,Z 516.216,A -85,B 0,C 180,E1 -24720.014,E2 -24720.014} C_VEL
LIN {X 0,Y 143.644,Z 523.078,A -85,B 0,C 180,E1 -24723.875,E2 -24723.875} C_VEL
LIN {X 0,Y 140.293,Z 528.569,A -85,B 0,C 180,E1 -24727.932,E2 -24727.932} C_VEL
LIN {X 0,Y 137.659,Z 532.875,A -85,B 0,C 180,E1 -24732.163,E2 -24732.163} C_VEL
LIN {X 0,Y 136.244,Z 535.152,A -85,B 0,C 180,E1 -24735.054,E2 -24735.054} C_VEL
LIN {X 0,Y 135.173,Z 537.001,A -85,B 0,C 180,E1 -24737.997,E2 -24737.997} C_VEL
LIN {X 0,Y 134.428,Z 538.386,A -85,B 0,C 180,E1 -24740.977,E2 -24740.977} C_VEL
LIN {X 0,Y 133.949,Z 539.371,A -85,B 0,C 180,E1 -24743.977,E2 -24743.977} C_VEL
LIN {X 0,Y 133.596,Z 540.112,A -85,B 0,C 180,E1 -24748.244,E2 -24748.244} C_VEL
LIN {X 0,Y 133.659,Z 540.005,A -85,B 0,C 180,E1 -24753.014,E2 -24753.014} C_VEL
LIN {X 0,Y 133.949,Z 539.419,A -85,B 0,C 180,E1 -24756.024,E2 -24756.024} C_VEL
LIN {X 0,Y 135.172,Z 537.096,A -85,B 0,C 180,E1 -24762.004,E2 -24762.004} C_VEL
LIN {X 0,Y 136.902,Z 534.226,A -85,B 0,C 180,E1 -24766.401,E2 -24766.401} C_VEL
LIN {X 0,Y 139.295,Z 530.333,A -85,B 0,C 180,E1 -24770.682,E2 -24770.682} C_VEL
LIN {X 0,Y 142.343,Z 525.308,A -85,B 0,C 180,E1 -24774.814,E2 -24774.814} C_VEL
LIN {X 0,Y 146.193,Z 518.972,A -85,B 0,C 180,E1 -24778.734,E2 -24778.734} C_VEL
LIN {X 0,Y 150.583,Z 510.704,A -85,B 0,C 180,E1 -24782.649,E2 -24782.649} C_VEL
LIN {X 0,Y 155.182,Z 501.199,A -85,B 0,C 180,E1 -24786.069,E2 -24786.069} C_VEL
LIN {X 0,Y 156.006,Z 499.276,A -85,B 0,C 180,E1 -24786.649,E2 -24786.649} C_VEL
LIN {X 0,Y 156.696,Z 493.19,A -85,B 0,C 180,E1 -24788.897,E2 -24788.897} C_VEL
LIN {X 0,Y 156.596,Z 484.699,A -85,B 0,C 180,E1 -24791.949,E2 -24791.949} C_VEL
LIN {X 0,Y 155.714,Z 476.962,A -85,B 0,C 180,E1 -24794.696,E2 -24794.696} C_VEL
LIN {X 0,Y 154.263,Z 471.245,A -85,B 0,C 180,E1 -24796.892,E2 -24796.892} C_VEL
LIN {X 0,Y 151.383,Z 463.54,A -85,B 0,C 180,E1 -24800.165,E2 -24800.165} C_VEL
LIN {X 0,Y 148.557,Z 457.465,A -85,B 0,C 180,E1 -24802.986,E2 -24802.986} C_VEL
LIN {X 0,Y 146.574,Z 453.873,A -85,B 0,C 180,E1 -24804.873,E2 -24804.873} C_VEL
LIN {X 0,Y 144.001,Z 449.98,A -85,B 0,C 180,E1 -24807.219,E2 -24807.219} C_VEL
LIN {X 0,Y 143.235,Z 448.828,A -85,B 0,C 180,E1 -24807.959,E2 -24807.959} C_VEL
LIN {X 0,Y 141.01,Z 446.129,A -85,B 0,C 180,E1 -24810.002,E2 -24810.002} C_VEL
LIN {X 0,Y 140.166,Z 444.077,A -85,B 0,C 180,E1 -24811.032,E2 -24811.032} C_VEL
LIN {X 0,Y 137.603,Z 442.067,A -85,B 0,C 180,E1 -24813.455,E2 -24813.455} C_VEL
LIN {X 0,Y 136.325,Z 439.636,A -85,B 0,C 180,E1 -24815.033,E2 -24815.033} C_VEL
LIN {X 0,Y 136.087,Z 438.529,A -85,B 0,C 180,E1 -24815.597,E2 -24815.597} C_VEL
LIN {X 0,Y 136.246,Z 438.514,A -85,B 0,C 180,E1 -24818.833,E2 -24818.833} C_VEL
LIN {X 0,Y 136.288,Z 438.506,A -85,B 0,C 180,E1 -24825.058,E2 -24825.058} C_VEL
LIN {X 0,Y 136.504,Z 438.479,A -85,B 0,C 180,E1 -24828.115,E2 -24828.115} C_VEL
LIN {X 0,Y 136.611,Z 438.465,A -85,B 0,C 180,E1 -24831.122,E2 -24831.122} C_VEL
LIN {X 0,Y 137.137,Z 438.4,A -85,B 0,C 180,E1 -24840,E2 -24840} C_VEL
LIN {X 0,Y 136.611,Z 438.468,A -85,B 0,C 180,E1 -24848.878,E2 -24848.878} C_VEL
LIN {X 0,Y 136.495,Z 438.484,A -85,B 0,C 180,E1 -24851.959,E2 -24851.959} C_VEL
LIN {X 0,Y 136.259,Z 438.51,A -85,B 0,C 180,E1 -24858.027,E2 -24858.027} C_VEL
LIN {X 0,Y 136.329,Z 439.288,A -85,B 0,C 180,E1 -24861.884,E2 -24861.884} C_VEL
LIN {X 0,Y 136.363,Z 440.136,A -85,B 0,C 180,E1 -24864.553,E2 -24864.553} C_VEL
LIN {X 0,Y 137.445,Z 442.857,A -85,B 0,C 180,E1 -24865.965,E2 -24865.965} C_VEL
LIN {X 0,Y 140.036,Z 446.121,A -85,B 0,C 180,E1 -24868.576,E2 -24868.576} C_VEL
LIN {X 0,Y 140.815,Z 447.096,A -85,B 0,C 180,E1 -24869.308,E2 -24869.308} C_VEL
LIN {X 0,Y 142.549,Z 450.702,A -85,B 0,C 180,E1 -24871.176,E2 -24871.176} C_VEL
LIN {X 0,Y 144.292,Z 453.042,A -85,B 0,C 180,E1 -24872.707,E2 -24872.707} C_VEL
LIN {X 0,Y 146.2,Z 456.904,A -85,B 0,C 180,E1 -24874.6,E2 -24874.6} C_VEL
LIN {X 0,Y 147.309,Z 459.233,A -85,B 0,C 180,E1 -24875.68,E2 -24875.68} C_VEL
LIN {X 0,Y 149.405,Z 463.657,A -85,B 0,C 180,E1 -24877.7,E2 -24877.7} C_VEL
LIN {X 0,Y 151.986,Z 469.944,A -85,B 0,C 180,E1 -24880.344,E2 -24880.344} C_VEL
LIN {X 0,Y 154.757,Z 478.818,A -85,B 0,C 180,E1 -24883.741,E2 -24883.741} C_VEL
LIN {X 0,Y 155.352,Z 484.095,A -85,B 0,C 180,E1 -24885.439,E2 -24885.439} C_VEL
LIN {X 0,Y 155.316,Z 492.729,A -85,B 0,C 180,E1 -24888.13,E2 -24888.13} C_VEL
LIN {X 0,Y 154.405,Z 502.218,A -85,B 0,C 180,E1 -24891.27,E2 -24891.27} C_VEL
LIN {X 0,Y 152.91,Z 510.05,A -85,B 0,C 180,E1 -24894.125,E2 -24894.125} C_VEL
LIN {X 0,Y 149.85,Z 516.723,A -85,B 0,C 180,E1 -24896.559,E2 -24896.559} C_VEL
LIN {X 0,Y 145.276,Z 525.419,A -85,B 0,C 180,E1 -24900.55,E2 -24900.55} C_VEL
LIN {X 0,Y 141.746,Z 531.652,A -85,B 0,C 180,E1 -24904.288,E2 -24904.288} C_VEL
LIN {X 0,Y 138.132,Z 537.746,A -85,B 0,C 180,E1 -24909.136,E2 -24909.136} C_VEL
LIN {X 0,Y 135.872,Z 541.713,A -85,B 0,C 180,E1 -24913.471,E2 -24913.471} C_VEL
LIN {X 0,Y 134.437,Z 544.651,A -85,B 0,C 180,E1 -24917.929,E2 -24917.929} C_VEL
LIN {X 0,Y 133.824,Z 546.05,A -85,B 0,C 180,E1 -24920.935,E2 -24920.935} C_VEL
LIN {X 0,Y 133.398,Z 547.663,A -85,B 0,C 180,E1 -24926.98,E2 -24926.98} C_VEL
LIN {X 0,Y 133.532,Z 547.879,A -85,B 0,C 180,E1 -24930,E2 -24930} C_VEL
LIN {X 0,Y 133.398,Z 547.648,A -85,B 0,C 180,E1 -24933.02,E2 -24933.02} C_VEL
LIN {X 0,Y 133.824,Z 546.016,A -85,B 0,C 180,E1 -24939.064,E2 -24939.064} C_VEL
LIN {X 0,Y 134.436,Z 544.603,A -85,B 0,C 180,E1 -24942.07,E2 -24942.07} C_VEL
LIN {X 0,Y 135.871,Z 541.644,A -85,B 0,C 180,E1 -24946.528,E2 -24946.528} C_VEL
LIN {X 0,Y 138.132,Z 537.651,A -85,B 0,C 180,E1 -24950.864,E2 -24950.864} C_VEL
LIN {X 0,Y 141.745,Z 531.519,A -85,B 0,C 180,E1 -24955.711,E2 -24955.711} C_VEL
LIN {X 0,Y 145.401,Z 525.077,A -85,B 0,C 180,E1 -24959.537,E2 -24959.537} C_VEL
LIN {X 0,Y 149.848,Z 516.526,A -85,B 0,C 180,E1 -24963.441,E2 -24963.441} C_VEL
LIN {X 0,Y 152.866,Z 509.811,A -85,B 0,C 180,E1 -24965.886,E2 -24965.886} C_VEL
LIN {X 0,Y 154.494,Z 500.928,A -85,B 0,C 180,E1 -24969.089,E2 -24969.089} C_VEL
LIN {X 0,Y 155.336,Z 490.651,A -85,B 0,C 180,E1 -24972.436,E2 -24972.436} C_VEL
LIN {X 0,Y 155.208,Z 482.399,A -85,B 0,C 180,E1 -24974.968,E2 -24974.968} C_VEL
LIN {X 0,Y 154.206,Z 476.79,A -85,B 0,C 180,E1 -24976.872,E2 -24976.872} C_VEL
LIN {X 0,Y 150.618,Z 466.516,A -85,B 0,C 180,E1 -24980.906,E2 -24980.906} C_VEL
LIN {X 0,Y 146.132,Z 456.784,A -85,B 0,C 180,E1 -24985.277,E2 -24985.277} C_VEL
LIN {X 0,Y 144.216,Z 452.889,A -85,B 0,C 180,E1 -24987.17,E2 -24987.17} C_VEL
LIN {X 0,Y 143.691,Z 452.07,A -85,B 0,C 180,E1 -24987.642,E2 -24987.642} C_VEL
LIN {X 0,Y 139.505,Z 448.979,A -85,B 0,C 180,E1 -24991.036,E2 -24991.036} C_VEL
LIN {X 0,Y 132.613,Z 445.182,A -85,B 0,C 180,E1 -24997.795,E2 -24997.795} C_VEL
LIN {X 0,Y 131.394,Z 444.088,A -85,B 0,C 180,E1 -24999.365,E2 -24999.365} C_VEL
LIN {X 0,Y 129.664,Z 441.152,A -85,B 0,C 180,E1 -25002.249,E2 -25002.249} C_VEL
LIN {X 0,Y 129.209,Z 439.541,A -85,B 0,C 180,E1 -25003.408,E2 -25003.408} C_VEL
LIN {X 0,Y 129.419,Z 439.364,A -85,B 0,C 180,E1 -25007.815,E2 -25007.815} C_VEL
LIN {X 0,Y 129.532,Z 439.349,A -85,B 0,C 180,E1 -25010.632,E2 -25010.632} C_VEL
LIN {X 0,Y 130.092,Z 439.278,A -85,B 0,C 180,E1 -25020,E2 -25020} C_VEL
LIN {X 0,Y 129.532,Z 439.35,A -85,B 0,C 180,E1 -25029.368,E2 -25029.368} C_VEL
LIN {X 0,Y 129.395,Z 439.367,A -85,B 0,C 180,E1 -25032.548,E2 -25032.548} C_VEL
LIN {X 0,Y 129.207,Z 439.44,A -85,B 0,C 180,E1 -25037.306,E2 -25037.306} C_VEL
LIN {X 0,Y 130.073,Z 442.093,A -85,B 0,C 180,E1 -25039.224,E2 -25039.224} C_VEL
LIN {X 0,Y 132.649,Z 444.722,A -85,B 0,C 180,E1 -25042.887,E2 -25042.887} C_VEL
LIN {X 0,Y 133.552,Z 445.342,A -85,B 0,C 180,E1 -25043.966,E2 -25043.966} C_VEL
LIN {X 0,Y 135.073,Z 448.449,A -85,B 0,C 180,E1 -25046.145,E2 -25046.145} C_VEL
LIN {X 0,Y 137.293,Z 450.701,A -85,B 0,C 180,E1 -25048.575,E2 -25048.575} C_VEL
LIN {X 0,Y 138.81,Z 453.565,A -85,B 0,C 180,E1 -25050.418,E2 -25050.418} C_VEL
LIN {X 0,Y 140.035,Z 454.935,A -85,B 0,C 180,E1 -25051.632,E2 -25051.632} C_VEL
LIN {X 0,Y 143.31,Z 460.751,A -85,B 0,C 180,E1 -25055.214,E2 -25055.214} C_VEL
LIN {X 0,Y 146.309,Z 467.277,A -85,B 0,C 180,E1 -25058.643,E2 -25058.643} C_VEL
LIN {X 0,Y 148.807,Z 474.557,A -85,B 0,C 180,E1 -25061.98,E2 -25061.98} C_VEL
LIN {X 0,Y 150.165,Z 480.802,A -85,B 0,C 180,E1 -25064.59,E2 -25064.59} C_VEL
LIN {X 0,Y 150.668,Z 486.918,A -85,B 0,C 180,E1 -25066.938,E2 -25066.938} C_VEL
LIN {X 0,Y 150.522,Z 494.998,A -85,B 0,C 180,E1 -25070.059,E2 -25070.059} C_VEL
LIN {X 0,Y 150.081,Z 499.016,A -85,B 0,C 180,E1 -25071.65,E2 -25071.65} C_VEL
LIN {X 0,Y 149.592,Z 500.944,A -85,B 0,C 180,E1 -25072.356,E2 -25072.356} C_VEL
LIN {X 0,Y 145.144,Z 509.899,A -85,B 0,C 180,E1 -25075.601,E2 -25075.601} C_VEL
LIN {X 0,Y 140.81,Z 517.648,A -85,B 0,C 180,E1 -25079.23,E2 -25079.23} C_VEL
LIN {X 0,Y 137.295,Z 523.284,A -85,B 0,C 180,E1 -25082.568,E2 -25082.568} C_VEL
LIN {X 0,Y 133.732,Z 528.775,A -85,B 0,C 180,E1 -25086.788,E2 -25086.788} C_VEL
LIN {X 0,Y 130.916,Z 533.08,A -85,B 0,C 180,E1 -25091.21,E2 -25091.21} C_VEL
LIN {X 0,Y 129.39,Z 535.357,A -85,B 0,C 180,E1 -25094.242,E2 -25094.242} C_VEL
LIN {X 0,Y 128.237,Z 537.205,A -85,B 0,C 180,E1 -25097.337,E2 -25097.337} C_VEL
LIN {X 0,Y 127.414,Z 538.591,A -85,B 0,C 180,E1 -25100.475,E2 -25100.475} C_VEL
LIN {X 0,Y 126.889,Z 539.576,A -85,B 0,C 180,E1 -25103.64,E2 -25103.64} C_VEL
LIN {X 0,Y 126.585,Z 540.18,A -85,B 0,C 180,E1 -25106.818,E2 -25106.818} C_VEL
LIN {X 0,Y 126.505,Z 540.405,A -85,B 0,C 180,E1 -25110,E2 -25110} C_VEL
LIN {X 0,Y 126.585,Z 540.209,A -85,B 0,C 180,E1 -25113.183,E2 -25113.183} C_VEL
LIN {X 0,Y 126.889,Z 539.623,A -85,B 0,C 180,E1 -25116.36,E2 -25116.36} C_VEL
LIN {X 0,Y 128.236,Z 537.3,A -85,B 0,C 180,E1 -25122.664,E2 -25122.664} C_VEL
LIN {X 0,Y 130.089,Z 534.43,A -85,B 0,C 180,E1 -25127.286,E2 -25127.286} C_VEL
LIN {X 0,Y 132.673,Z 530.536,A -85,B 0,C 180,E1 -25131.766,E2 -25131.766} C_VEL
LIN {X 0,Y 135.928,Z 525.511,A -85,B 0,C 180,E1 -25136.071,E2 -25136.071} C_VEL
LIN {X 0,Y 140.006,Z 519.174,A -85,B 0,C 180,E1 -25140.131,E2 -25140.131} C_VEL
LIN {X 0,Y 144.402,Z 511.376,A -85,B 0,C 180,E1 -25143.967,E2 -25143.967} C_VEL
LIN {X 0,Y 148.594,Z 503.179,A -85,B 0,C 180,E1 -25147.088,E2 -25147.088} C_VEL
LIN {X 0,Y 150.134,Z 499.485,A -85,B 0,C 180,E1 -25148.335,E2 -25148.335} C_VEL
LIN {X 0,Y 150.782,Z 492.106,A -85,B 0,C 180,E1 -25151.259,E2 -25151.259} C_VEL
LIN {X 0,Y 150.616,Z 483.855,A -85,B 0,C 180,E1 -25154.421,E2 -25154.421} C_VEL
LIN {X 0,Y 149.647,Z 477.478,A -85,B 0,C 180,E1 -25156.956,E2 -25156.956} C_VEL
LIN {X 0,Y 147.295,Z 469.702,A -85,B 0,C 180,E1 -25160.436,E2 -25160.436} C_VEL
LIN {X 0,Y 144.118,Z 462.3,A -85,B 0,C 180,E1 -25164.184,E2 -25164.184} C_VEL
LIN {X 0,Y 141.593,Z 457.787,A -85,B 0,C 180,E1 -25166.908,E2 -25166.908} C_VEL
LIN {X 0,Y 140.333,Z 455.367,A -85,B 0,C 180,E1 -25168.362,E2 -25168.362} C_VEL
LIN {X 0,Y 137.836,Z 451.959,A -85,B 0,C 180,E1 -25171.027,E2 -25171.027} C_VEL
LIN {X 0,Y 137.028,Z 450.267,A -85,B 0,C 180,E1 -25172.095,E2 -25172.095} C_VEL
LIN {X 0,Y 134.696,Z 447.874,A -85,B 0,C 180,E1 -25174.71,E2 -25174.71} C_VEL
LIN {X 0,Y 133.35,Z 445.07,A -85,B 0,C 180,E1 -25176.717,E2 -25176.717} C_VEL
LIN {X 0,Y 130.517,Z 442.743,A -85,B 0,C 180,E1 -25180.538,E2 -25180.538} C_VEL
LIN {X 0,Y 129.316,Z 440.039,A -85,B 0,C 180,E1 -25182.913,E2 -25182.913} C_VEL
LIN {X 0,Y 129.192,Z 439.391,A -85,B 0,C 180,E1 -25183.405,E2 -25183.405} C_VEL
LIN {X 0,Y 129.421,Z 439.361,A -85,B 0,C 180,E1 -25187.815,E2 -25187.815} C_VEL
LIN {X 0,Y 129.533,Z 439.347,A -85,B 0,C 180,E1 -25190.632,E2 -25190.632} C_VEL
LIN {X 0,Y 130.093,Z 439.278,A -85,B 0,C 180,E1 -25200,E2 -25200} C_VEL
LIN {X 0,Y 129.533,Z 439.351,A -85,B 0,C 180,E1 -25209.368,E2 -25209.368} C_VEL
LIN {X 0,Y 129.397,Z 439.366,A -85,B 0,C 180,E1 -25212.548,E2 -25212.548} C_VEL
LIN {X 0,Y 129.219,Z 439.592,A -85,B 0,C 180,E1 -25216.286,E2 -25216.286} C_VEL
LIN {X 0,Y 129.969,Z 441.803,A -85,B 0,C 180,E1 -25217.911,E2 -25217.911} C_VEL
LIN {X 0,Y 132.151,Z 444.909,A -85,B 0,C 180,E1 -25221.314,E2 -25221.314} C_VEL
LIN {X 0,Y 133.893,Z 446.647,A -85,B 0,C 180,E1 -25223.49,E2 -25223.49} C_VEL
LIN {X 0,Y 135.751,Z 450.576,A -85,B 0,C 180,E1 -25226.107,E2 -25226.107} C_VEL
LIN {X 0,Y 137.645,Z 452.998,A -85,B 0,C 180,E1 -25228.183,E2 -25228.183} C_VEL
LIN {X 0,Y 139.659,Z 457.101,A -85,B 0,C 180,E1 -25230.615,E2 -25230.615} C_VEL
LIN {X 0,Y 140.948,Z 459.459,A -85,B 0,C 180,E1 -25232.041,E2 -25232.041} C_VEL
LIN {X 0,Y 144.213,Z 466.676,A -85,B 0,C 180,E1 -25235.789,E2 -25235.789} C_VEL
LIN {X 0,Y 147.085,Z 474.289,A -85,B 0,C 180,E1 -25239.281,E2 -25239.281} C_VEL
LIN {X 0,Y 149.243,Z 482.086,A -85,B 0,C 180,E1 -25242.537,E2 -25242.537} C_VEL
LIN {X 0,Y 149.672,Z 485.283,A -85,B 0,C 180,E1 -25243.7,E2 -25243.7} C_VEL
LIN {X 0,Y 149.444,Z 494.301,A -85,B 0,C 180,E1 -25246.715,E2 -25246.715} C_VEL
LIN {X 0,Y 148.331,Z 503.255,A -85,B 0,C 180,E1 -25249.877,E2 -25249.877} C_VEL
LIN {X 0,Y 146.969,Z 509.84,A -85,B 0,C 180,E1 -25252.432,E2 -25252.432} C_VEL
LIN {X 0,Y 145.643,Z 513.311,A -85,B 0,C 180,E1 -25253.763,E2 -25253.763} C_VEL
LIN {X 0,Y 140.729,Z 522.369,A -85,B 0,C 180,E1 -25257.615,E2 -25257.615} C_VEL
LIN {X 0,Y 136.685,Z 529.416,A -85,B 0,C 180,E1 -25261.6,E2 -25261.6} C_VEL
LIN {X 0,Y 133.569,Z 534.262,A -85,B 0,C 180,E1 -25265.106,E2 -25265.106} C_VEL
LIN {X 0,Y 130.581,Z 538.977,A -85,B 0,C 180,E1 -25269.522,E2 -25269.522} C_VEL
LIN {X 0,Y 128.448,Z 542.585,A -85,B 0,C 180,E1 -25274.123,E2 -25274.123} C_VEL
LIN {X 0,Y 127.466,Z 544.447,A -85,B 0,C 180,E1 -25277.259,E2 -25277.259} C_VEL
LIN {X 0,Y 126.793,Z 545.845,A -85,B 0,C 180,E1 -25280.428,E2 -25280.428} C_VEL
LIN {X 0,Y 126.412,Z 546.846,A -85,B 0,C 180,E1 -25283.616,E2 -25283.616} C_VEL
LIN {X 0,Y 126.303,Z 547.458,A -85,B 0,C 180,E1 -25286.81,E2 -25286.81} C_VEL
LIN {X 0,Y 126.428,Z 547.675,A -85,B 0,C 180,E1 -25290,E2 -25290} C_VEL
LIN {X 0,Y 126.303,Z 547.443,A -85,B 0,C 180,E1 -25293.189,E2 -25293.189} C_VEL
LIN {X 0,Y 126.412,Z 546.821,A -85,B 0,C 180,E1 -25296.384,E2 -25296.384} C_VEL
LIN {X 0,Y 126.793,Z 545.811,A -85,B 0,C 180,E1 -25299.572,E2 -25299.572} C_VEL
LIN {X 0,Y 127.466,Z 544.397,A -85,B 0,C 180,E1 -25302.741,E2 -25302.741} C_VEL
LIN {X 0,Y 129.05,Z 541.438,A -85,B 0,C 180,E1 -25307.429,E2 -25307.429} C_VEL
LIN {X 0,Y 131.499,Z 537.445,A -85,B 0,C 180,E1 -25311.969,E2 -25311.969} C_VEL
LIN {X 0,Y 135.379,Z 531.313,A -85,B 0,C 180,E1 -25317.016,E2 -25317.016} C_VEL
LIN {X 0,Y 139.957,Z 523.63,A -85,B 0,C 180,E1 -25321.651,E2 -25321.651} C_VEL
LIN {X 0,Y 143.946,Z 516.318,A -85,B 0,C 180,E1 -25325.007,E2 -25325.007} C_VEL
LIN {X 0,Y 146.375,Z 511.395,A -85,B 0,C 180,E1 -25326.882,E2 -25326.882} C_VEL
LIN {X 0,Y 147.942,Z 504.924,A -85,B 0,C 180,E1 -25329.397,E2 -25329.397} C_VEL
LIN {X 0,Y 149.243,Z 495.161,A -85,B 0,C 180,E1 -25332.906,E2 -25332.906} C_VEL
LIN {X 0,Y 149.646,Z 488.18,A -85,B 0,C 180,E1 -25335.214,E2 -25335.214} C_VEL
LIN {X 0,Y 149.367,Z 483.13,A -85,B 0,C 180,E1 -25336.951,E2 -25336.951} C_VEL
LIN {X 0,Y 147.762,Z 476.702,A -85,B 0,C 180,E1 -25339.553,E2 -25339.553} C_VEL
LIN {X 0,Y 144.636,Z 467.719,A -85,B 0,C 180,E1 -25343.539,E2 -25343.539} C_VEL
LIN {X 0,Y 141.635,Z 461.083,A -85,B 0,C 180,E1 -25346.919,E2 -25346.919} C_VEL
LIN {X 0,Y 139.729,Z 457.114,A -85,B 0,C 180,E1 -25349.113,E2 -25349.113} C_VEL
LIN {X 0,Y 137.806,Z 453.471,A -85,B 0,C 180,E1 -25351.334,E2 -25351.334} C_VEL
LIN {X 0,Y 137.147,Z 452.285,A -85,B 0,C 180,E1 -25352.121,E2 -25352.121} C_VEL
LIN {X 0,Y 134.704,Z 448.872,A -85,B 0,C 180,E1 -25354.918,E2 -25354.918} C_VEL
LIN {X 0,Y 133.6,Z 446.319,A -85,B 0,C 180,E1 -25356.558,E2 -25356.558} C_VEL
LIN {X 0,Y 131.394,Z 444.088,A -85,B 0,C 180,E1 -25359.365,E2 -25359.365} C_VEL
LIN {X 0,Y 129.626,Z 442.992,A -85,B 0,C 180,E1 -25361.8,E2 -25361.8} C_VEL
LIN {X 0,Y 126.768,Z 443.237,A -85,B 0,C 180,E1 -25366.06,E2 -25366.06} C_VEL
LIN {X 0,Y 124.907,Z 443.875,A -85,B 0,C 180,E1 -25369.624,E2 -25369.624} C_VEL
LIN {X 0,Y 123.951,Z 443.76,A -85,B 0,C 180,E1 -25372.359,E2 -25372.359} C_VEL
LIN {X 0,Y 123.741,Z 443.499,A -85,B 0,C 180,E1 -25373.273,E2 -25373.273} C_VEL
LIN {X 0,Y 123.245,Z 441.209,A -85,B 0,C 180,E1 -25380,E2 -25380} C_VEL
LIN {X 0,Y 127.171,Z 446.469,A -85,B 0,C 180,E1 -25396.556,E2 -25396.556} C_VEL
LIN {X 0,Y 128.202,Z 449.118,A -85,B 0,C 180,E1 -25398.996,E2 -25398.996} C_VEL
LIN {X 0,Y 130.929,Z 451.966,A -85,B 0,C 180,E1 -25403.216,E2 -25403.216} C_VEL
LIN {X 0,Y 132.264,Z 454.706,A -85,B 0,C 180,E1 -25405.403,E2 -25405.403} C_VEL
LIN {X 0,Y 134.31,Z 457.452,A -85,B 0,C 180,E1 -25408.096,E2 -25408.096} C_VEL
LIN {X 0,Y 137.036,Z 461.978,A -85,B 0,C 180,E1 -25411.588,E2 -25411.588} C_VEL
LIN {X 0,Y 139.944,Z 467.657,A -85,B 0,C 180,E1 -25415.277,E2 -25415.277} C_VEL
LIN {X 0,Y 142.44,Z 474.399,A -85,B 0,C 180,E1 -25418.892,E2 -25418.892} C_VEL
LIN {X 0,Y 144.237,Z 481.466,A -85,B 0,C 180,E1 -25422.3,E2 -25422.3} C_VEL
LIN {X 0,Y 144.876,Z 488.262,A -85,B 0,C 180,E1 -25425.19,E2 -25425.19} C_VEL
LIN {X 0,Y 144.584,Z 496.013,A -85,B 0,C 180,E1 -25428.41,E2 -25428.41} C_VEL
LIN {X 0,Y 143.856,Z 501.158,A -85,B 0,C 180,E1 -25430.572,E2 -25430.572} C_VEL
LIN {X 0,Y 140.08,Z 508.769,A -85,B 0,C 180,E1 -25433.393,E2 -25433.393} C_VEL
LIN {X 0,Y 135.536,Z 516.628,A -85,B 0,C 180,E1 -25437.013,E2 -25437.013} C_VEL
LIN {X 0,Y 131.036,Z 523.49,A -85,B 0,C 180,E1 -25441.138,E2 -25441.138} C_VEL
LIN {X 0,Y 127.235,Z 528.98,A -85,B 0,C 180,E1 -25445.527,E2 -25445.527} C_VEL
LIN {X 0,Y 124.197,Z 533.285,A -85,B 0,C 180,E1 -25450.152,E2 -25450.152} C_VEL
LIN {X 0,Y 122.572,Z 535.562,A -85,B 0,C 180,E1 -25453.341,E2 -25453.341} C_VEL
LIN {X 0,Y 121.33,Z 537.41,A -85,B 0,C 180,E1 -25456.603,E2 -25456.603} C_VEL
LIN {X 0,Y 120.429,Z 538.795,A -85,B 0,C 180,E1 -25459.917,E2 -25459.917} C_VEL
LIN {X 0,Y 119.84,Z 539.78,A -85,B 0,C 180,E1 -25463.265,E2 -25463.265} C_VEL
LIN {X 0,Y 119.498,Z 540.384,A -85,B 0,C 180,E1 -25466.629,E2 -25466.629} C_VEL
LIN {X 0,Y 119.419,Z 540.609,A -85,B 0,C 180,E1 -25470,E2 -25470} C_VEL
LIN {X 0,Y 119.498,Z 540.413,A -85,B 0,C 180,E1 -25473.372,E2 -25473.372} C_VEL
LIN {X 0,Y 119.841,Z 539.826,A -85,B 0,C 180,E1 -25476.736,E2 -25476.736} C_VEL
LIN {X 0,Y 121.328,Z 537.503,A -85,B 0,C 180,E1 -25483.398,E2 -25483.398} C_VEL
LIN {X 0,Y 123.31,Z 534.634,A -85,B 0,C 180,E1 -25488.269,E2 -25488.269} C_VEL
LIN {X 0,Y 126.085,Z 530.739,A -85,B 0,C 180,E1 -25492.966,E2 -25492.966} C_VEL
LIN {X 0,Y 129.589,Z 525.714,A -85,B 0,C 180,E1 -25497.451,E2 -25497.451} C_VEL
LIN {X 0,Y 133.903,Z 519.376,A -85,B 0,C 180,E1 -25501.659,E2 -25501.659} C_VEL
LIN {X 0,Y 138.304,Z 512.048,A -85,B 0,C 180,E1 -25505.401,E2 -25505.401} C_VEL
LIN {X 0,Y 142.995,Z 503.38,A -85,B 0,C 180,E1 -25508.804,E2 -25508.804} C_VEL
LIN {X 0,Y 143.85,Z 501.605,A -85,B 0,C 180,E1 -25509.43,E2 -25509.43} C_VEL
LIN {X 0,Y 144.784,Z 494.946,A -85,B 0,C 180,E1 -25512.22,E2 -25512.22} C_VEL
LIN {X 0,Y 144.874,Z 486.37,A -85,B 0,C 180,E1 -25515.787,E2 -25515.787} C_VEL
LIN {X 0,Y 143.987,Z 479.92,A -85,B 0,C 180,E1 -25518.641,E2 -25518.641} C_VEL
LIN {X 0,Y 142.17,Z 473.423,A -85,B 0,C 180,E1 -25521.837,E2 -25521.837} C_VEL
LIN {X 0,Y 139.566,Z 466.879,A -85,B 0,C 180,E1 -25525.493,E2 -25525.493} C_VEL
LIN {X 0,Y 136.808,Z 461.377,A -85,B 0,C 180,E1 -25529.088,E2 -25529.088} C_VEL
LIN {X 0,Y 134.525,Z 457.873,A -85,B 0,C 180,E1 -25531.953,E2 -25531.953} C_VEL
LIN {X 0,Y 133.934,Z 456.442,A -85,B 0,C 180,E1 -25532.902,E2 -25532.902} C_VEL
LIN {X 0,Y 132.36,Z 454.817,A -85,B 0,C 180,E1 -25534.863,E2 -25534.863} C_VEL
LIN {X 0,Y 130.787,Z 451.601,A -85,B 0,C 180,E1 -25537.488,E2 -25537.488} C_VEL
LIN {X 0,Y 128.263,Z 449.161,A -85,B 0,C 180,E1 -25541.428,E2 -25541.428} C_VEL
LIN {X 0,Y 127.057,Z 446.153,A -85,B 0,C 180,E1 -25544.356,E2 -25544.356} C_VEL
LIN {X 0,Y 123.459,Z 441.827,A -85,B 0,C 180,E1 -25560,E2 -25560} C_VEL
LIN {X 0,Y 127.258,Z 446.359,A -85,B 0,C 180,E1 -25575.31,E2 -25575.31} C_VEL
LIN {X 0,Y 128.837,Z 450.124,A -85,B 0,C 180,E1 -25578.898,E2 -25578.898} C_VEL
LIN {X 0,Y 131.218,Z 453.044,A -85,B 0,C 180,E1 -25582.537,E2 -25582.537} C_VEL
LIN {X 0,Y 132.738,Z 456.517,A -85,B 0,C 180,E1 -25585.06,E2 -25585.06} C_VEL
LIN {X 0,Y 134.407,Z 459.095,A -85,B 0,C 180,E1 -25587.262,E2 -25587.262} C_VEL
LIN {X 0,Y 135.906,Z 462.499,A -85,B 0,C 180,E1 -25589.424,E2 -25589.424} C_VEL
LIN {X 0,Y 137.028,Z 464.614,A -85,B 0,C 180,E1 -25590.856,E2 -25590.856} C_VEL
LIN {X 0,Y 139.616,Z 471.144,A -85,B 0,C 180,E1 -25594.493,E2 -25594.493} C_VEL
LIN {X 0,Y 142.097,Z 478.518,A -85,B 0,C 180,E1 -25598.186,E2 -25598.186} C_VEL
LIN {X 0,Y 143.792,Z 485.547,A -85,B 0,C 180,E1 -25601.375,E2 -25601.375} C_VEL
LIN {X 0,Y 144.014,Z 490.042,A -85,B 0,C 180,E1 -25603.095,E2 -25603.095} C_VEL
LIN {X 0,Y 143.371,Z 497.765,A -85,B 0,C 180,E1 -25605.903,E2 -25605.903} C_VEL
LIN {X 0,Y 141.843,Z 506.642,A -85,B 0,C 180,E1 -25609.34,E2 -25609.34} C_VEL
LIN {X 0,Y 140.603,Z 511.43,A -85,B 0,C 180,E1 -25611.331,E2 -25611.331} C_VEL
LIN {X 0,Y 138.162,Z 516.317,A -85,B 0,C 180,E1 -25613.294,E2 -25613.294} C_VEL
LIN {X 0,Y 133.324,Z 524.583,A -85,B 0,C 180,E1 -25617.294,E2 -25617.294} C_VEL
LIN {X 0,Y 129.094,Z 531.246,A -85,B 0,C 180,E1 -25621.552,E2 -25621.552} C_VEL
LIN {X 0,Y 124.925,Z 537.339,A -85,B 0,C 180,E1 -25626.808,E2 -25626.808} C_VEL
LIN {X 0,Y 122.248,Z 541.304,A -85,B 0,C 180,E1 -25631.567,E2 -25631.567} C_VEL
LIN {X 0,Y 120.525,Z 544.243,A -85,B 0,C 180,E1 -25636.511,E2 -25636.511} C_VEL
LIN {X 0,Y 119.785,Z 545.641,A -85,B 0,C 180,E1 -25639.862,E2 -25639.862} C_VEL
LIN {X 0,Y 119.219,Z 547.255,A -85,B 0,C 180,E1 -25646.62,E2 -25646.62} C_VEL
LIN {X 0,Y 119.333,Z 547.471,A -85,B 0,C 180,E1 -25650,E2 -25650} C_VEL
LIN {X 0,Y 119.219,Z 547.239,A -85,B 0,C 180,E1 -25653.379,E2 -25653.379} C_VEL
LIN {X 0,Y 119.785,Z 545.606,A -85,B 0,C 180,E1 -25660.137,E2 -25660.137} C_VEL
LIN {X 0,Y 120.525,Z 544.192,A -85,B 0,C 180,E1 -25663.488,E2 -25663.488} C_VEL
LIN {X 0,Y 122.247,Z 541.232,A -85,B 0,C 180,E1 -25668.433,E2 -25668.433} C_VEL
LIN {X 0,Y 124.925,Z 537.24,A -85,B 0,C 180,E1 -25673.191,E2 -25673.191} C_VEL
LIN {X 0,Y 129.093,Z 531.108,A -85,B 0,C 180,E1 -25678.448,E2 -25678.448} C_VEL
LIN {X 0,Y 133.327,Z 524.413,A -85,B 0,C 180,E1 -25682.704,E2 -25682.704} C_VEL
LIN {X 0,Y 138.161,Z 516.111,A -85,B 0,C 180,E1 -25686.705,E2 -25686.705} C_VEL
LIN {X 0,Y 140.561,Z 511.181,A -85,B 0,C 180,E1 -25688.682,E2 -25688.682} C_VEL
LIN {X 0,Y 142.238,Z 504.132,A -85,B 0,C 180,E1 -25691.582,E2 -25691.582} C_VEL
LIN {X 0,Y 143.674,Z 494.524,A -85,B 0,C 180,E1 -25695.174,E2 -25695.174} C_VEL
LIN {X 0,Y 143.976,Z 487.923,A -85,B 0,C 180,E1 -25697.541,E2 -25697.541} C_VEL
LIN {X 0,Y 143.133,Z 482.677,A -85,B 0,C 180,E1 -25699.753,E2 -25699.753} C_VEL
LIN {X 0,Y 141.018,Z 475.21,A -85,B 0,C 180,E1 -25703.27,E2 -25703.27} C_VEL
LIN {X 0,Y 138.021,Z 467.133,A -85,B 0,C 180,E1 -25707.508,E2 -25707.508} C_VEL
LIN {X 0,Y 136.362,Z 463.128,A -85,B 0,C 180,E1 -25709.834,E2 -25709.834} C_VEL
LIN {X 0,Y 133.971,Z 458.217,A -85,B 0,C 180,E1 -25713.101,E2 -25713.101} C_VEL
LIN {X 0,Y 131.687,Z 454.57,A -85,B 0,C 180,E1 -25716.197,E2 -25716.197} C_VEL
LIN {X 0,Y 130.827,Z 452.522,A -85,B 0,C 180,E1 -25717.704,E2 -25717.704} C_VEL
LIN {X 0,Y 127.881,Z 448.447,A -85,B 0,C 180,E1 -25722.51,E2 -25722.51} C_VEL
LIN {X 0,Y 127.178,Z 446.192,A -85,B 0,C 180,E1 -25724.372,E2 -25724.372} C_VEL
LIN {X 0,Y 123.741,Z 443.499,A -85,B 0,C 180,E1 -25733.273,E2 -25733.273} C_VEL
LIN {X 0,Y 123.369,Z 443.251,A -85,B 0,C 180,E1 -25735.085,E2 -25735.085} C_VEL
LIN {X 0,Y 122.992,Z 443.666,A -85,B 0,C 180,E1 -25736.901,E2 -25736.901} C_VEL
LIN {X 0,Y 122.33,Z 445.76,A -85,B 0,C 180,E1 -25740.48,E2 -25740.48} C_VEL
LIN {X 0,Y 121.948,Z 449.703,A -85,B 0,C 180,E1 -25745.918,E2 -25745.918} C_VEL
LIN {X 0,Y 122.164,Z 450.555,A -85,B 0,C 180,E1 -25747.783,E2 -25747.783} C_VEL
LIN {X 0,Y 124.825,Z 453.097,A -85,B 0,C 180,E1 -25755.721,E2 -25755.721} C_VEL
LIN {X 0,Y 125.542,Z 455.25,A -85,B 0,C 180,E1 -25757.884,E2 -25757.884} C_VEL
LIN {X 0,Y 128.079,Z 458.552,A -85,B 0,C 180,E1 -25762.589,E2 -25762.589} C_VEL
LIN {X 0,Y 130.809,Z 463.265,A -85,B 0,C 180,E1 -25767.173,E2 -25767.173} C_VEL
LIN {X 0,Y 133.278,Z 467.869,A -85,B 0,C 180,E1 -25770.94,E2 -25770.94} C_VEL
LIN {X 0,Y 135.752,Z 473.318,A -85,B 0,C 180,E1 -25774.714,E2 -25774.714} C_VEL
LIN {X 0,Y 137.759,Z 479.921,A -85,B 0,C 180,E1 -25778.481,E2 -25778.481} C_VEL
LIN {X 0,Y 138.94,Z 486.275,A -85,B 0,C 180,E1 -25781.747,E2 -25781.747} C_VEL
LIN {X 0,Y 139.074,Z 492.229,A -85,B 0,C 180,E1 -25784.456,E2 -25784.456} C_VEL
LIN {X 0,Y 138.374,Z 499.795,A -85,B 0,C 180,E1 -25787.875,E2 -25787.875} C_VEL
LIN {X 0,Y 137.6,Z 503.16,A -85,B 0,C 180,E1 -25789.367,E2 -25789.367} C_VEL
LIN {X 0,Y 133.068,Z 511.296,A -85,B 0,C 180,E1 -25792.596,E2 -25792.596} C_VEL
LIN {X 0,Y 127.982,Z 519.286,A -85,B 0,C 180,E1 -25796.692,E2 -25796.692} C_VEL
LIN {X 0,Y 123.41,Z 525.693,A -85,B 0,C 180,E1 -25801.049,E2 -25801.049} C_VEL
LIN {X 0,Y 119.643,Z 530.769,A -85,B 0,C 180,E1 -25805.721,E2 -25805.721} C_VEL
LIN {X 0,Y 116.602,Z 534.71,A -85,B 0,C 180,E1 -25810.64,E2 -25810.64} C_VEL
LIN {X 0,Y 114.427,Z 537.615,A -85,B 0,C 180,E1 -25815.779,E2 -25815.779} C_VEL
LIN {X 0,Y 113.432,Z 539,A -85,B 0,C 180,E1 -25819.288,E2 -25819.288} C_VEL
LIN {X 0,Y 112.79,Z 539.984,A -85,B 0,C 180,E1 -25822.841,E2 -25822.841} C_VEL
LIN {X 0,Y 112.424,Z 540.588,A -85,B 0,C 180,E1 -25826.416,E2 -25826.416} C_VEL
LIN {X 0,Y 112.335,Z 540.812,A -85,B 0,C 180,E1 -25830,E2 -25830} C_VEL
LIN {X 0,Y 112.424,Z 540.616,A -85,B 0,C 180,E1 -25833.584,E2 -25833.584} C_VEL
LIN {X 0,Y 112.79,Z 540.03,A -85,B 0,C 180,E1 -25837.159,E2 -25837.159} C_VEL
LIN {X 0,Y 114.425,Z 537.707,A -85,B 0,C 180,E1 -25844.222,E2 -25844.222} C_VEL
LIN {X 0,Y 116.578,Z 534.837,A -85,B 0,C 180,E1 -25849.365,E2 -25849.365} C_VEL
LIN {X 0,Y 119.557,Z 530.943,A -85,B 0,C 180,E1 -25854.299,E2 -25854.299} C_VEL
LIN {X 0,Y 123.338,Z 525.916,A -85,B 0,C 180,E1 -25858.97,E2 -25858.97} C_VEL
LIN {X 0,Y 127.908,Z 519.578,A -85,B 0,C 180,E1 -25863.33,E2 -25863.33} C_VEL
LIN {X 0,Y 132.307,Z 512.712,A -85,B 0,C 180,E1 -25866.971,E2 -25866.971} C_VEL
LIN {X 0,Y 137.505,Z 503.582,A -85,B 0,C 180,E1 -25870.668,E2 -25870.668} C_VEL
LIN {X 0,Y 138.169,Z 501.816,A -85,B 0,C 180,E1 -25871.396,E2 -25871.396} C_VEL
LIN {X 0,Y 139.013,Z 495.17,A -85,B 0,C 180,E1 -25874.417,E2 -25874.417} C_VEL
LIN {X 0,Y 139.178,Z 487.997,A -85,B 0,C 180,E1 -25877.658,E2 -25877.658} C_VEL
LIN {X 0,Y 138.311,Z 482.154,A -85,B 0,C 180,E1 -25880.566,E2 -25880.566} C_VEL
LIN {X 0,Y 136.769,Z 476.334,A -85,B 0,C 180,E1 -25883.776,E2 -25883.776} C_VEL
LIN {X 0,Y 134.518,Z 470.208,A -85,B 0,C 180,E1 -25887.62,E2 -25887.62} C_VEL
LIN {X 0,Y 133.019,Z 467.131,A -85,B 0,C 180,E1 -25889.872,E2 -25889.872} C_VEL
LIN {X 0,Y 130.061,Z 462.012,A -85,B 0,C 180,E1 -25894.387,E2 -25894.387} C_VEL
LIN {X 0,Y 127.45,Z 457.603,A -85,B 0,C 180,E1 -25898.996,E2 -25898.996} C_VEL
LIN {X 0,Y 125.796,Z 455.645,A -85,B 0,C 180,E1 -25902.103,E2 -25902.103} C_VEL
LIN {X 0,Y 124.698,Z 452.801,A -85,B 0,C 180,E1 -25905.308,E2 -25905.308} C_VEL
LIN {X 0,Y 121.925,Z 448.855,A -85,B 0,C 180,E1 -25920,E2 -25920} C_VEL
LIN {X 0,Y 125.041,Z 453.098,A -85,B 0,C 180,E1 -25934.547,E2 -25934.547} C_VEL
LIN {X 0,Y 126.239,Z 456.268,A -85,B 0,C 180,E1 -25937.83,E2 -25937.83} C_VEL
LIN {X 0,Y 127.977,Z 458.661,A -85,B 0,C 180,E1 -25941,E2 -25941} C_VEL
LIN {X 0,Y 129.501,Z 462.368,A -85,B 0,C 180,E1 -25944.018,E2 -25944.018} C_VEL
LIN {X 0,Y 130.491,Z 463.905,A -85,B 0,C 180,E1 -25945.522,E2 -25945.522} C_VEL
LIN {X 0,Y 133.193,Z 470.396,A -85,B 0,C 180,E1 -25950.084,E2 -25950.084} C_VEL
LIN {X 0,Y 135.326,Z 476.643,A -85,B 0,C 180,E1 -25953.804,E2 -25953.804} C_VEL
LIN {X 0,Y 137.405,Z 484.293,A -85,B 0,C 180,E1 -25957.863,E2 -25957.863} C_VEL
LIN {X 0,Y 138.476,Z 490.204,A -85,B 0,C 180,E1 -25960.754,E2 -25960.754} C_VEL
LIN {X 0,Y 137.804,Z 497.9,A -85,B 0,C 180,E1 -25963.774,E2 -25963.774} C_VEL
LIN {X 0,Y 135.878,Z 507.602,A -85,B 0,C 180,E1 -25967.747,E2 -25967.747} C_VEL
LIN {X 0,Y 134.262,Z 512.9,A -85,B 0,C 180,E1 -25970.116,E2 -25970.116} C_VEL
LIN {X 0,Y 129.832,Z 520.466,A -85,B 0,C 180,E1 -25973.455,E2 -25973.455} C_VEL
LIN {X 0,Y 125.082,Z 527.777,A -85,B 0,C 180,E1 -25977.641,E2 -25977.641} C_VEL
LIN {X 0,Y 120.776,Z 533.855,A -85,B 0,C 180,E1 -25982.255,E2 -25982.255} C_VEL
LIN {X 0,Y 117.349,Z 538.57,A -85,B 0,C 180,E1 -25987.09,E2 -25987.09} C_VEL
LIN {X 0,Y 114.775,Z 542.176,A -85,B 0,C 180,E1 -25992.171,E2 -25992.171} C_VEL
LIN {X 0,Y 113.616,Z 544.039,A -85,B 0,C 180,E1 -25995.674,E2 -25995.674} C_VEL
LIN {X 0,Y 112.777,Z 545.437,A -85,B 0,C 180,E1 -25999.225,E2 -25999.225} C_VEL
LIN {X 0,Y 112.127,Z 547.051,A -85,B 0,C 180,E1 -26006.406,E2 -26006.406} C_VEL
LIN {X 0,Y 112.25,Z 547.267,A -85,B 0,C 180,E1 -26010,E2 -26010} C_VEL
LIN {X 0,Y 112.127,Z 547.035,A -85,B 0,C 180,E1 -26013.593,E2 -26013.593} C_VEL
LIN {X 0,Y 112.777,Z 545.401,A -85,B 0,C 180,E1 -26020.775,E2 -26020.775} C_VEL
LIN {X 0,Y 113.616,Z 543.987,A -85,B 0,C 180,E1 -26024.325,E2 -26024.325} C_VEL
LIN {X 0,Y 115.498,Z 541.026,A -85,B 0,C 180,E1 -26029.552,E2 -26029.552} C_VEL
LIN {X 0,Y 118.416,Z 537.034,A -85,B 0,C 180,E1 -26034.547,E2 -26034.547} C_VEL
LIN {X 0,Y 122.893,Z 530.902,A -85,B 0,C 180,E1 -26040.026,E2 -26040.026} C_VEL
LIN {X 0,Y 127.371,Z 524.206,A -85,B 0,C 180,E1 -26044.441,E2 -26044.441} C_VEL
LIN {X 0,Y 132.526,Z 515.904,A -85,B 0,C 180,E1 -26048.544,E2 -26048.544} C_VEL
LIN {X 0,Y 134.223,Z 512.668,A -85,B 0,C 180,E1 -26049.898,E2 -26049.898} C_VEL
LIN {X 0,Y 136.3,Z 505.158,A -85,B 0,C 180,E1 -26053.194,E2 -26053.194} C_VEL
LIN {X 0,Y 137.926,Z 496.133,A -85,B 0,C 180,E1 -26056.804,E2 -26056.804} C_VEL
LIN {X 0,Y 138.347,Z 490.095,A -85,B 0,C 180,E1 -26059.19,E2 -26059.19} C_VEL
LIN {X 0,Y 137.294,Z 484.078,A -85,B 0,C 180,E1 -26062.101,E2 -26062.101} C_VEL
LIN {X 0,Y 135.087,Z 476.082,A -85,B 0,C 180,E1 -26066.347,E2 -26066.347} C_VEL
LIN {X 0,Y 132.642,Z 468.867,A -85,B 0,C 180,E1 -26070.652,E2 -26070.652} C_VEL
LIN {X 0,Y 130.306,Z 463.68,A -85,B 0,C 180,E1 -26074.439,E2 -26074.439} C_VEL
LIN {X 0,Y 127.709,Z 458.407,A -85,B 0,C 180,E1 -26079.043,E2 -26079.043} C_VEL
LIN {X 0,Y 125.403,Z 454.628,A -85,B 0,C 180,E1 -26083.622,E2 -26083.622} C_VEL
LIN {X 0,Y 124.872,Z 452.829,A -85,B 0,C 180,E1 -26085.329,E2 -26085.329} C_VEL
LIN {X 0,Y 121.732,Z 448.266,A -85,B 0,C 180,E1 -26100,E2 -26100} C_VEL
LIN {X 0,Y 122.164,Z 450.555,A -85,B 0,C 180,E1 -26107.783,E2 -26107.783} C_VEL
LIN {X 0,Y 122.381,Z 451.712,A -85,B 0,C 180,E1 -26109.546,E2 -26109.546} C_VEL
LIN {X 0,Y 122.393,Z 455.156,A -85,B 0,C 180,E1 -26112.207,E2 -26112.207} C_VEL
LIN {X 0,Y 122.373,Z 459.787,A -85,B 0,C 180,E1 -26115.353,E2 -26115.353} C_VEL
LIN {X 0,Y 122.578,Z 460.991,A -85,B 0,C 180,E1 -26116.483,E2 -26116.483} C_VEL
LIN {X 0,Y 124.742,Z 464.443,A -85,B 0,C 180,E1 -26121.482,E2 -26121.482} C_VEL
LIN {X 0,Y 127.1,Z 468.968,A -85,B 0,C 180,E1 -26126.255,E2 -26126.255} C_VEL
LIN {X 0,Y 129.235,Z 473.468,A -85,B 0,C 180,E1 -26130.201,E2 -26130.201} C_VEL
LIN {X 0,Y 131.1,Z 478.152,A -85,B 0,C 180,E1 -26133.707,E2 -26133.707} C_VEL
LIN {X 0,Y 132.595,Z 484.003,A -85,B 0,C 180,E1 -26137.34,E2 -26137.34} C_VEL
LIN {X 0,Y 133.443,Z 490.313,A -85,B 0,C 180,E1 -26140.859,E2 -26140.859} C_VEL
LIN {X 0,Y 133.207,Z 496.322,A -85,B 0,C 180,E1 -26143.825,E2 -26143.825} C_VEL
LIN {X 0,Y 132.056,Z 503.376,A -85,B 0,C 180,E1 -26147.269,E2 -26147.269} C_VEL
LIN {X 0,Y 130.373,Z 506.822,A -85,B 0,C 180,E1 -26148.673,E2 -26148.673} C_VEL
LIN {X 0,Y 124.712,Z 515.717,A -85,B 0,C 180,E1 -26152.714,E2 -26152.714} C_VEL
LIN {X 0,Y 119.625,Z 522.876,A -85,B 0,C 180,E1 -26157.082,E2 -26157.082} C_VEL
LIN {X 0,Y 115.756,Z 527.705,A -85,B 0,C 180,E1 -26160.941,E2 -26160.941} C_VEL
LIN {X 0,Y 112.029,Z 532.389,A -85,B 0,C 180,E1 -26165.935,E2 -26165.935} C_VEL
LIN {X 0,Y 109.045,Z 535.972,A -85,B 0,C 180,E1 -26171.201,E2 -26171.201} C_VEL
LIN {X 0,Y 107.562,Z 537.819,A -85,B 0,C 180,E1 -26174.85,E2 -26174.85} C_VEL
LIN {X 0,Y 106.455,Z 539.205,A -85,B 0,C 180,E1 -26178.577,E2 -26178.577} C_VEL
LIN {X 0,Y 105.745,Z 540.189,A -85,B 0,C 180,E1 -26182.362,E2 -26182.362} C_VEL
LIN {X 0,Y 105.344,Z 540.792,A -85,B 0,C 180,E1 -26186.175,E2 -26186.175} C_VEL
LIN {X 0,Y 105.238,Z 541.016,A -85,B 0,C 180,E1 -26190,E2 -26190} C_VEL
LIN {X 0,Y 105.344,Z 540.82,A -85,B 0,C 180,E1 -26193.826,E2 -26193.826} C_VEL
LIN {X 0,Y 105.745,Z 540.234,A -85,B 0,C 180,E1 -26197.639,E2 -26197.639} C_VEL
LIN {X 0,Y 107.56,Z 537.91,A -85,B 0,C 180,E1 -26205.151,E2 -26205.151} C_VEL
LIN {X 0,Y 109.901,Z 535.041,A -85,B 0,C 180,E1 -26210.593,E2 -26210.593} C_VEL
LIN {X 0,Y 113.102,Z 531.146,A -85,B 0,C 180,E1 -26215.784,E2 -26215.784} C_VEL
LIN {X 0,Y 117.186,Z 526.118,A -85,B 0,C 180,E1 -26220.649,E2 -26220.649} C_VEL
LIN {X 0,Y 122.034,Z 519.781,A -85,B 0,C 180,E1 -26225.164,E2 -26225.164} C_VEL
LIN {X 0,Y 127.484,Z 511.659,A -85,B 0,C 180,E1 -26229.484,E2 -26229.484} C_VEL
LIN {X 0,Y 132.066,Z 503.789,A -85,B 0,C 180,E1 -26232.727,E2 -26232.727} C_VEL
LIN {X 0,Y 133.244,Z 496.691,A -85,B 0,C 180,E1 -26236.222,E2 -26236.222} C_VEL
LIN {X 0,Y 133.566,Z 490.886,A -85,B 0,C 180,E1 -26239.059,E2 -26239.059} C_VEL
LIN {X 0,Y 133.044,Z 486.161,A -85,B 0,C 180,E1 -26241.648,E2 -26241.648} C_VEL
LIN {X 0,Y 131.8,Z 480.434,A -85,B 0,C 180,E1 -26245.103,E2 -26245.103} C_VEL
LIN {X 0,Y 129.877,Z 474.77,A -85,B 0,C 180,E1 -26249.066,E2 -26249.066} C_VEL
LIN {X 0,Y 127.321,Z 469.268,A -85,B 0,C 180,E1 -26253.794,E2 -26253.794} C_VEL
LIN {X 0,Y 124.955,Z 464.811,A -85,B 0,C 180,E1 -26258.556,E2 -26258.556} C_VEL
LIN {X 0,Y 122.828,Z 461.533,A -85,B 0,C 180,E1 -26263.376,E2 -26263.376} C_VEL
LIN {X 0,Y 122.424,Z 460.1,A -85,B 0,C 180,E1 -26265.029,E2 -26265.029} C_VEL
LIN {X 0,Y 121.888,Z 459.214,A -85,B 0,C 180,E1 -26266.665,E2 -26266.665} C_VEL
LIN {X 0,Y 120.008,Z 455.785,A -85,B 0,C 180,E1 -26280,E2 -26280} C_VEL
LIN {X 0,Y 122.32,Z 459.448,A -85,B 0,C 180,E1 -26293.287,E2 -26293.287} C_VEL
LIN {X 0,Y 123.951,Z 463.383,A -85,B 0,C 180,E1 -26298.171,E2 -26298.171} C_VEL
LIN {X 0,Y 124.704,Z 464.539,A -85,B 0,C 180,E1 -26299.764,E2 -26299.764} C_VEL
LIN {X 0,Y 127.219,Z 470.689,A -85,B 0,C 180,E1 -26305.349,E2 -26305.349} C_VEL
LIN {X 0,Y 129.21,Z 476.317,A -85,B 0,C 180,E1 -26309.509,E2 -26309.509} C_VEL
LIN {X 0,Y 131.145,Z 483.337,A -85,B 0,C 180,E1 -26313.909,E2 -26313.909} C_VEL
LIN {X 0,Y 132.321,Z 489.132,A -85,B 0,C 180,E1 -26317.183,E2 -26317.183} C_VEL
LIN {X 0,Y 132.898,Z 493.249,A -85,B 0,C 180,E1 -26319.39,E2 -26319.39} C_VEL
LIN {X 0,Y 132.209,Z 499.131,A -85,B 0,C 180,E1 -26321.907,E2 -26321.907} C_VEL
LIN {X 0,Y 130.302,Z 507.384,A -85,B 0,C 180,E1 -26325.478,E2 -26325.478} C_VEL
LIN {X 0,Y 128.671,Z 512.69,A -85,B 0,C 180,E1 -26328.002,E2 -26328.002} C_VEL
LIN {X 0,Y 127.04,Z 515.913,A -85,B 0,C 180,E1 -26329.456,E2 -26329.456} C_VEL
LIN {X 0,Y 121.543,Z 524.176,A -85,B 0,C 180,E1 -26333.651,E2 -26333.651} C_VEL
LIN {X 0,Y 116.784,Z 530.841,A -85,B 0,C 180,E1 -26338.225,E2 -26338.225} C_VEL
LIN {X 0,Y 111.985,Z 536.932,A -85,B 0,C 180,E1 -26343.94,E2 -26343.94} C_VEL
LIN {X 0,Y 108.808,Z 540.896,A -85,B 0,C 180,E1 -26349.191,E2 -26349.191} C_VEL
LIN {X 0,Y 106.706,Z 543.834,A -85,B 0,C 180,E1 -26354.724,E2 -26354.724} C_VEL
LIN {X 0,Y 105.797,Z 545.233,A -85,B 0,C 180,E1 -26358.504,E2 -26358.504} C_VEL
LIN {X 0,Y 105.036,Z 546.847,A -85,B 0,C 180,E1 -26366.163,E2 -26366.163} C_VEL
LIN {X 0,Y 105.168,Z 547.064,A -85,B 0,C 180,E1 -26370,E2 -26370} C_VEL
LIN {X 0,Y 105.035,Z 546.83,A -85,B 0,C 180,E1 -26373.836,E2 -26373.836} C_VEL
LIN {X 0,Y 105.797,Z 545.196,A -85,B 0,C 180,E1 -26381.495,E2 -26381.495} C_VEL
LIN {X 0,Y 106.705,Z 543.781,A -85,B 0,C 180,E1 -26385.275,E2 -26385.275} C_VEL
LIN {X 0,Y 108.808,Z 540.82,A -85,B 0,C 180,E1 -26390.808,E2 -26390.808} C_VEL
LIN {X 0,Y 111.984,Z 536.828,A -85,B 0,C 180,E1 -26396.06,E2 -26396.06} C_VEL
LIN {X 0,Y 116.784,Z 530.696,A -85,B 0,C 180,E1 -26401.774,E2 -26401.774} C_VEL
LIN {X 0,Y 121.542,Z 523.999,A -85,B 0,C 180,E1 -26406.348,E2 -26406.348} C_VEL
LIN {X 0,Y 127.035,Z 515.697,A -85,B 0,C 180,E1 -26410.545,E2 -26410.545} C_VEL
LIN {X 0,Y 128.604,Z 512.451,A -85,B 0,C 180,E1 -26412.024,E2 -26412.024} C_VEL
LIN {X 0,Y 130.881,Z 504.456,A -85,B 0,C 180,E1 -26415.728,E2 -26415.728} C_VEL
LIN {X 0,Y 132.448,Z 496.672,A -85,B 0,C 180,E1 -26419.014,E2 -26419.014} C_VEL
LIN {X 0,Y 132.775,Z 493.091,A -85,B 0,C 180,E1 -26420.567,E2 -26420.567} C_VEL
LIN {X 0,Y 131.579,Z 485.466,A -85,B 0,C 180,E1 -26424.673,E2 -26424.673} C_VEL
LIN {X 0,Y 129.374,Z 476.983,A -85,B 0,C 180,E1 -26429.835,E2 -26429.835} C_VEL
LIN {X 0,Y 128.234,Z 473.568,A -85,B 0,C 180,E1 -26432.233,E2 -26432.233} C_VEL
LIN {X 0,Y 126.709,Z 469.397,A -85,B 0,C 180,E1 -26435.418,E2 -26435.418} C_VEL
LIN {X 0,Y 124.488,Z 464.35,A -85,B 0,C 180,E1 -26440.2,E2 -26440.2} C_VEL
LIN {X 0,Y 123.089,Z 461.922,A -85,B 0,C 180,E1 -26443.412,E2 -26443.412} C_VEL
LIN {X 0,Y 122.607,Z 460.364,A -85,B 0,C 180,E1 -26445.052,E2 -26445.052} C_VEL
LIN {X 0,Y 122.065,Z 459.293,A -85,B 0,C 180,E1 -26446.685,E2 -26446.685} C_VEL
LIN {X 0,Y 119.834,Z 455.23,A -85,B 0,C 180,E1 -26460,E2 -26460} C_VEL
LIN {X 0,Y 122.22,Z 459.659,A -85,B 0,C 180,E1 -26474.997,E2 -26474.997} C_VEL
LIN {X 0,Y 122.578,Z 460.991,A -85,B 0,C 180,E1 -26476.483,E2 -26476.483} C_VEL
LIN {X 0,Y 123.093,Z 463.731,A -85,B 0,C 180,E1 -26478.929,E2 -26478.929} C_VEL
LIN {X 0,Y 123.435,Z 469.479,A -85,B 0,C 180,E1 -26482.698,E2 -26482.698} C_VEL
LIN {X 0,Y 124.091,Z 476.336,A -85,B 0,C 180,E1 -26487.238,E2 -26487.238} C_VEL
LIN {X 0,Y 124.733,Z 478.161,A -85,B 0,C 180,E1 -26488.84,E2 -26488.84} C_VEL
LIN {X 0,Y 126.418,Z 483.21,A -85,B 0,C 180,E1 -26492.918,E2 -26492.918} C_VEL
LIN {X 0,Y 127.414,Z 488.336,A -85,B 0,C 180,E1 -26496.367,E2 -26496.367} C_VEL
LIN {X 0,Y 127.896,Z 493.841,A -85,B 0,C 180,E1 -26499.708,E2 -26499.708} C_VEL
LIN {X 0,Y 127.374,Z 499.148,A -85,B 0,C 180,E1 -26502.552,E2 -26502.552} C_VEL
LIN {X 0,Y 126.038,Z 505.351,A -85,B 0,C 180,E1 -26505.812,E2 -26505.812} C_VEL
LIN {X 0,Y 121.429,Z 512.696,A -85,B 0,C 180,E1 -26509.004,E2 -26509.004} C_VEL
LIN {X 0,Y 116.365,Z 519.699,A -85,B 0,C 180,E1 -26512.846,E2 -26512.846} C_VEL
LIN {X 0,Y 111.209,Z 526.103,A -85,B 0,C 180,E1 -26517.509,E2 -26517.509} C_VEL
LIN {X 0,Y 106.819,Z 531.181,A -85,B 0,C 180,E1 -26522.577,E2 -26522.577} C_VEL
LIN {X 0,Y 103.313,Z 535.119,A -85,B 0,C 180,E1 -26528.029,E2 -26528.029} C_VEL
LIN {X 0,Y 100.715,Z 538.025,A -85,B 0,C 180,E1 -26533.792,E2 -26533.792} C_VEL
LIN {X 0,Y 99.512,Z 539.409,A -85,B 0,C 180,E1 -26537.768,E2 -26537.768} C_VEL
LIN {X 0,Y 98.703,Z 540.393,A -85,B 0,C 180,E1 -26541.813,E2 -26541.813} C_VEL
LIN {X 0,Y 98.259,Z 540.996,A -85,B 0,C 180,E1 -26545.899,E2 -26545.899} C_VEL
LIN {X 0,Y 98.152,Z 541.22,A -85,B 0,C 180,E1 -26550,E2 -26550} C_VEL
LIN {X 0,Y 98.259,Z 541.024,A -85,B 0,C 180,E1 -26554.102,E2 -26554.102} C_VEL
LIN {X 0,Y 98.703,Z 540.438,A -85,B 0,C 180,E1 -26558.188,E2 -26558.188} C_VEL
LIN {X 0,Y 100.711,Z 538.114,A -85,B 0,C 180,E1 -26566.209,E2 -26566.209} C_VEL
LIN {X 0,Y 103.288,Z 535.244,A -85,B 0,C 180,E1 -26571.978,E2 -26571.978} C_VEL
LIN {X 0,Y 106.736,Z 531.35,A -85,B 0,C 180,E1 -26577.447,E2 -26577.447} C_VEL
LIN {X 0,Y 111.148,Z 526.32,A -85,B 0,C 180,E1 -26582.512,E2 -26582.512} C_VEL
LIN {X 0,Y 116.297,Z 519.983,A -85,B 0,C 180,E1 -26587.18,E2 -26587.18} C_VEL
LIN {X 0,Y 121.685,Z 512.441,A -85,B 0,C 180,E1 -26591.338,E2 -26591.338} C_VEL
LIN {X 0,Y 125.977,Z 505.76,A -85,B 0,C 180,E1 -26594.215,E2 -26594.215} C_VEL
LIN {X 0,Y 127.198,Z 500.889,A -85,B 0,C 180,E1 -26596.744,E2 -26596.744} C_VEL
LIN {X 0,Y 127.978,Z 494.323,A -85,B 0,C 180,E1 -26600.249,E2 -26600.249} C_VEL
LIN {X 0,Y 127.557,Z 488.648,A -85,B 0,C 180,E1 -26603.681,E2 -26603.681} C_VEL
LIN {X 0,Y 126.525,Z 483.446,A -85,B 0,C 180,E1 -26607.209,E2 -26607.209} C_VEL
LIN {X 0,Y 125.124,Z 479.062,A -85,B 0,C 180,E1 -26610.706,E2 -26610.706} C_VEL
LIN {X 0,Y 123.396,Z 474.828,A -85,B 0,C 180,E1 -26614.712,E2 -26614.712} C_VEL
LIN {X 0,Y 121.396,Z 470.55,A -85,B 0,C 180,E1 -26619.674,E2 -26619.674} C_VEL
LIN {X 0,Y 119.352,Z 466.066,A -85,B 0,C 180,E1 -26626.376,E2 -26626.376} C_VEL
LIN {X 0,Y 117.509,Z 463.328,A -85,B 0,C 180,E1 -26636.571,E2 -26636.571} C_VEL
LIN {X 0,Y 117.678,Z 462.549,A -85,B 0,C 180,E1 -26640,E2 -26640} C_VEL
LIN {X 0,Y 118.748,Z 465.233,A -85,B 0,C 180,E1 -26650.227,E2 -26650.227} C_VEL
LIN {X 0,Y 119.76,Z 466.577,A -85,B 0,C 180,E1 -26653.576,E2 -26653.576} C_VEL
LIN {X 0,Y 121.255,Z 470.339,A -85,B 0,C 180,E1 -26658.589,E2 -26658.589} C_VEL
LIN {X 0,Y 123.233,Z 475.947,A -85,B 0,C 180,E1 -26664.148,E2 -26664.148} C_VEL
LIN {X 0,Y 124.861,Z 481.517,A -85,B 0,C 180,E1 -26668.583,E2 -26668.583} C_VEL
LIN {X 0,Y 126.384,Z 488.844,A -85,B 0,C 180,E1 -26673.474,E2 -26673.474} C_VEL
LIN {X 0,Y 127.211,Z 495.36,A -85,B 0,C 180,E1 -26677.424,E2 -26677.424} C_VEL
LIN {X 0,Y 126.952,Z 498.903,A -85,B 0,C 180,E1 -26679.191,E2 -26679.191} C_VEL
LIN {X 0,Y 125.373,Z 505.599,A -85,B 0,C 180,E1 -26682.274,E2 -26682.274} C_VEL
LIN {X 0,Y 123.163,Z 512.476,A -85,B 0,C 180,E1 -26685.651,E2 -26685.651} C_VEL
LIN {X 0,Y 121.682,Z 515.709,A -85,B 0,C 180,E1 -26687.262,E2 -26687.262} C_VEL
LIN {X 0,Y 115.853,Z 523.972,A -85,B 0,C 180,E1 -26691.552,E2 -26691.552} C_VEL
LIN {X 0,Y 110.772,Z 530.637,A -85,B 0,C 180,E1 -26696.278,E2 -26696.278} C_VEL
LIN {X 0,Y 105.64,Z 536.729,A -85,B 0,C 180,E1 -26702.244,E2 -26702.244} C_VEL
LIN {X 0,Y 102.185,Z 540.692,A -85,B 0,C 180,E1 -26707.773,E2 -26707.773} C_VEL
LIN {X 0,Y 99.83,Z 543.629,A -85,B 0,C 180,E1 -26713.644,E2 -26713.644} C_VEL
LIN {X 0,Y 98.813,Z 545.028,A -85,B 0,C 180,E1 -26717.679,E2 -26717.679} C_VEL
LIN {X 0,Y 98.186,Z 546.03,A -85,B 0,C 180,E1 -26721.769,E2 -26721.769} C_VEL
LIN {X 0,Y 97.942,Z 546.643,A -85,B 0,C 180,E1 -26725.885,E2 -26725.885} C_VEL
LIN {X 0,Y 98.074,Z 546.86,A -85,B 0,C 180,E1 -26730,E2 -26730} C_VEL
LIN {X 0,Y 97.942,Z 546.626,A -85,B 0,C 180,E1 -26734.115,E2 -26734.115} C_VEL
LIN {X 0,Y 98.186,Z 546.003,A -85,B 0,C 180,E1 -26738.23,E2 -26738.23} C_VEL
LIN {X 0,Y 98.812,Z 544.991,A -85,B 0,C 180,E1 -26742.32,E2 -26742.32} C_VEL
LIN {X 0,Y 99.83,Z 543.575,A -85,B 0,C 180,E1 -26746.355,E2 -26746.355} C_VEL
LIN {X 0,Y 102.185,Z 540.615,A -85,B 0,C 180,E1 -26752.227,E2 -26752.227} C_VEL
LIN {X 0,Y 105.639,Z 536.623,A -85,B 0,C 180,E1 -26757.755,E2 -26757.755} C_VEL
LIN {X 0,Y 110.774,Z 530.489,A -85,B 0,C 180,E1 -26763.72,E2 -26763.72} C_VEL
LIN {X 0,Y 115.852,Z 523.791,A -85,B 0,C 180,E1 -26768.448,E2 -26768.448} C_VEL
LIN {X 0,Y 121.673,Z 515.489,A -85,B 0,C 180,E1 -26772.741,E2 -26772.741} C_VEL
LIN {X 0,Y 123.737,Z 510.523,A -85,B 0,C 180,E1 -26775.232,E2 -26775.232} C_VEL
LIN {X 0,Y 126.478,Z 500.756,A -85,B 0,C 180,E1 -26779.82,E2 -26779.82} C_VEL
LIN {X 0,Y 127.132,Z 497.012,A -85,B 0,C 180,E1 -26781.544,E2 -26781.544} C_VEL
LIN {X 0,Y 126.795,Z 491.963,A -85,B 0,C 180,E1 -26784.409,E2 -26784.409} C_VEL
LIN {X 0,Y 125.577,Z 484.998,A -85,B 0,C 180,E1 -26788.822,E2 -26788.822} C_VEL
LIN {X 0,Y 124.127,Z 479.064,A -85,B 0,C 180,E1 -26793.067,E2 -26793.067} C_VEL
LIN {X 0,Y 122.883,Z 475.008,A -85,B 0,C 180,E1 -26796.4,E2 -26796.4} C_VEL
LIN {X 0,Y 121.056,Z 470.125,A -85,B 0,C 180,E1 -26801.379,E2 -26801.379} C_VEL
LIN {X 0,Y 119.566,Z 466.283,A -85,B 0,C 180,E1 -26806.402,E2 -26806.402} C_VEL
LIN {X 0,Y 117.54,Z 462.039,A -85,B 0,C 180,E1 -26820,E2 -26820} C_VEL
LIN {X 0,Y 119.108,Z 465.811,A -85,B 0,C 180,E1 -26833.652,E2 -26833.652} C_VEL
LIN {X 0,Y 121.181,Z 470.247,A -85,B 0,C 180,E1 -26840.364,E2 -26840.364} C_VEL
LIN {X 0,Y 123.185,Z 474.548,A -85,B 0,C 180,E1 -26845.334,E2 -26845.334} C_VEL
LIN {X 0,Y 124.733,Z 478.161,A -85,B 0,C 180,E1 -26848.84,E2 -26848.84} C_VEL
LIN {X 0,Y 125.367,Z 480.073,A -85,B 0,C 180,E1 -26850.391,E2 -26850.391} C_VEL
LIN {X 0,Y 125.49,Z 483.744,A -85,B 0,C 180,E1 -26852.518,E2 -26852.518} C_VEL
LIN {X 0,Y 124.895,Z 487.922,A -85,B 0,C 180,E1 -26854.461,E2 -26854.461} C_VEL
LIN {X 0,Y 123.405,Z 493.881,A -85,B 0,C 180,E1 -26857.019,E2 -26857.019} C_VEL
LIN {X 0,Y 122.016,Z 499.45,A -85,B 0,C 180,E1 -26859.779,E2 -26859.779} C_VEL
LIN {X 0,Y 120.653,Z 505.574,A -85,B 0,C 180,E1 -26863.271,E2 -26863.271} C_VEL
LIN {X 0,Y 120.02,Z 507.238,A -85,B 0,C 180,E1 -26864.166,E2 -26864.166} C_VEL
LIN {X 0,Y 113.732,Z 516.13,A -85,B 0,C 180,E1 -26868.372,E2 -26868.372} C_VEL
LIN {X 0,Y 107.968,Z 523.288,A -85,B 0,C 180,E1 -26872.979,E2 -26872.979} C_VEL
LIN {X 0,Y 103.586,Z 528.116,A -85,B 0,C 180,E1 -26877.128,E2 -26877.128} C_VEL
LIN {X 0,Y 99.236,Z 532.8,A -85,B 0,C 180,E1 -26882.592,E2 -26882.592} C_VEL
LIN {X 0,Y 95.699,Z 536.382,A -85,B 0,C 180,E1 -26888.458,E2 -26888.458} C_VEL
LIN {X 0,Y 93.916,Z 538.229,A -85,B 0,C 180,E1 -26892.583,E2 -26892.583} C_VEL
LIN {X 0,Y 92.58,Z 539.614,A -85,B 0,C 180,E1 -26896.837,E2 -26896.837} C_VEL
LIN {X 0,Y 91.693,Z 540.597,A -85,B 0,C 180,E1 -26901.183,E2 -26901.183} C_VEL
LIN {X 0,Y 91.205,Z 541.2,A -85,B 0,C 180,E1 -26905.581,E2 -26905.581} C_VEL
LIN {X 0,Y 91.058,Z 541.424,A -85,B 0,C 180,E1 -26910,E2 -26910} C_VEL
LIN {X 0,Y 91.186,Z 541.227,A -85,B 0,C 180,E1 -26914.421,E2 -26914.421} C_VEL
LIN {X 0,Y 91.693,Z 540.641,A -85,B 0,C 180,E1 -26918.818,E2 -26918.818} C_VEL
LIN {X 0,Y 93.912,Z 538.317,A -85,B 0,C 180,E1 -26927.419,E2 -26927.419} C_VEL
LIN {X 0,Y 96.749,Z 535.447,A -85,B 0,C 180,E1 -26933.549,E2 -26933.549} C_VEL
LIN {X 0,Y 100.473,Z 531.553,A -85,B 0,C 180,E1 -26939.318,E2 -26939.318} C_VEL
LIN {X 0,Y 105.242,Z 526.523,A -85,B 0,C 180,E1 -26944.585,E2 -26944.585} C_VEL
LIN {X 0,Y 110.716,Z 520.185,A -85,B 0,C 180,E1 -26949.404,E2 -26949.404} C_VEL
LIN {X 0,Y 116.069,Z 513.17,A -85,B 0,C 180,E1 -26953.397,E2 -26953.397} C_VEL
LIN {X 0,Y 119.91,Z 507.609,A -85,B 0,C 180,E1 -26955.889,E2 -26955.889} C_VEL
LIN {X 0,Y 120.692,Z 505.973,A -85,B 0,C 180,E1 -26956.71,E2 -26956.71} C_VEL
LIN {X 0,Y 122.19,Z 498.962,A -85,B 0,C 180,E1 -26960.751,E2 -26960.751} C_VEL
LIN {X 0,Y 122.384,Z 494.579,A -85,B 0,C 180,E1 -26963.511,E2 -26963.511} C_VEL
LIN {X 0,Y 121.825,Z 489.242,A -85,B 0,C 180,E1 -26967.338,E2 -26967.338} C_VEL
LIN {X 0,Y 120.958,Z 485.213,A -85,B 0,C 180,E1 -26970.639,E2 -26970.639} C_VEL
LIN {X 0,Y 119.258,Z 480.269,A -85,B 0,C 180,E1 -26975.637,E2 -26975.637} C_VEL
LIN {X 0,Y 117.6,Z 476.197,A -85,B 0,C 180,E1 -26980.81,E2 -26980.81} C_VEL
LIN {X 0,Y 116.278,Z 472.989,A -85,B 0,C 180,E1 -26986.009,E2 -26986.009} C_VEL
LIN {X 0,Y 115.553,Z 471.608,A -85,B 0,C 180,E1 -26989.487,E2 -26989.487} C_VEL
LIN {X 0,Y 114.965,Z 469.18,A -85,B 0,C 180,E1 -27000,E2 -27000} C_VEL
LIN {X 0,Y 115.965,Z 471.878,A -85,B 0,C 180,E1 -27010.475,E2 -27010.475} C_VEL
LIN {X 0,Y 116.742,Z 473.601,A -85,B 0,C 180,E1 -27013.934,E2 -27013.934} C_VEL
LIN {X 0,Y 118.059,Z 477.421,A -85,B 0,C 180,E1 -27019.112,E2 -27019.112} C_VEL
LIN {X 0,Y 119.192,Z 481.709,A -85,B 0,C 180,E1 -27023.453,E2 -27023.453} C_VEL
LIN {X 0,Y 120.367,Z 486.845,A -85,B 0,C 180,E1 -27027.847,E2 -27027.847} C_VEL
LIN {X 0,Y 121.295,Z 493.428,A -85,B 0,C 180,E1 -27032.576,E2 -27032.576} C_VEL
LIN {X 0,Y 121.658,Z 498.658,A -85,B 0,C 180,E1 -27036.024,E2 -27036.024} C_VEL
LIN {X 0,Y 121.242,Z 501.852,A -85,B 0,C 180,E1 -27037.776,E2 -27037.776} C_VEL
LIN {X 0,Y 118.893,Z 509.426,A -85,B 0,C 180,E1 -27041.559,E2 -27041.559} C_VEL
LIN {X 0,Y 116.458,Z 515.503,A -85,B 0,C 180,E1 -27044.839,E2 -27044.839} C_VEL
LIN {X 0,Y 110.344,Z 523.769,A -85,B 0,C 180,E1 -27049.243,E2 -27049.243} C_VEL
LIN {X 0,Y 104.902,Z 530.433,A -85,B 0,C 180,E1 -27054.111,E2 -27054.111} C_VEL
LIN {X 0,Y 99.38,Z 536.525,A -85,B 0,C 180,E1 -27060.328,E2 -27060.328} C_VEL
LIN {X 0,Y 95.613,Z 540.488,A -85,B 0,C 180,E1 -27066.154,E2 -27066.154} C_VEL
LIN {X 0,Y 93.005,Z 543.425,A -85,B 0,C 180,E1 -27072.406,E2 -27072.406} C_VEL
LIN {X 0,Y 91.863,Z 544.824,A -85,B 0,C 180,E1 -27076.731,E2 -27076.731} C_VEL
LIN {X 0,Y 90.871,Z 546.439,A -85,B 0,C 180,E1 -27085.564,E2 -27085.564} C_VEL
LIN {X 0,Y 90.972,Z 546.656,A -85,B 0,C 180,E1 -27090,E2 -27090} C_VEL
LIN {X 0,Y 90.871,Z 546.422,A -85,B 0,C 180,E1 -27094.435,E2 -27094.435} C_VEL
LIN {X 0,Y 91.862,Z 544.785,A -85,B 0,C 180,E1 -27103.268,E2 -27103.268} C_VEL
LIN {X 0,Y 93.004,Z 543.369,A -85,B 0,C 180,E1 -27107.593,E2 -27107.593} C_VEL
LIN {X 0,Y 95.612,Z 540.409,A -85,B 0,C 180,E1 -27113.846,E2 -27113.846} C_VEL
LIN {X 0,Y 99.378,Z 536.417,A -85,B 0,C 180,E1 -27119.672,E2 -27119.672} C_VEL
LIN {X 0,Y 104.906,Z 530.282,A -85,B 0,C 180,E1 -27125.887,E2 -27125.887} C_VEL
LIN {X 0,Y 110.343,Z 523.584,A -85,B 0,C 180,E1 -27130.756,E2 -27130.756} C_VEL
LIN {X 0,Y 115.473,Z 516.773,A -85,B 0,C 180,E1 -27134.42,E2 -27134.42} C_VEL
LIN {X 0,Y 117.147,Z 513.664,A -85,B 0,C 180,E1 -27136.047,E2 -27136.047} C_VEL
LIN {X 0,Y 120.274,Z 504.885,A -85,B 0,C 180,E1 -27140.596,E2 -27140.596} C_VEL
LIN {X 0,Y 121.499,Z 500.077,A -85,B 0,C 180,E1 -27142.965,E2 -27142.965} C_VEL
LIN {X 0,Y 121.352,Z 494.64,A -85,B 0,C 180,E1 -27146.395,E2 -27146.395} C_VEL
LIN {X 0,Y 120.501,Z 488.079,A -85,B 0,C 180,E1 -27151.026,E2 -27151.026} C_VEL
LIN {X 0,Y 119.543,Z 483.437,A -85,B 0,C 180,E1 -27154.771,E2 -27154.771} C_VEL
LIN {X 0,Y 118.85,Z 480.452,A -85,B 0,C 180,E1 -27157.396,E2 -27157.396} C_VEL
LIN {X 0,Y 117.393,Z 475.788,A -85,B 0,C 180,E1 -27162.582,E2 -27162.582} C_VEL
LIN {X 0,Y 116.578,Z 473.315,A -85,B 0,C 180,E1 -27166.046,E2 -27166.046} C_VEL
LIN {X 0,Y 115.741,Z 471.674,A -85,B 0,C 180,E1 -27169.504,E2 -27169.504} C_VEL
LIN {X 0,Y 114.852,Z 468.68,A -85,B 0,C 180,E1 -27180,E2 -27180} C_VEL
LIN {X 0,Y 115.317,Z 471.379,A -85,B 0,C 180,E1 -27190.535,E2 -27190.535} C_VEL
LIN {X 0,Y 116.211,Z 473.006,A -85,B 0,C 180,E1 -27194.622,E2 -27194.622} C_VEL
LIN {X 0,Y 117.895,Z 477.19,A -85,B 0,C 180,E1 -27200.958,E2 -27200.958} C_VEL
LIN {X 0,Y 119.062,Z 479.996,A -85,B 0,C 180,E1 -27204.406,E2 -27204.406} C_VEL
LIN {X 0,Y 120.693,Z 484.639,A -85,B 0,C 180,E1 -27209.138,E2 -27209.138} C_VEL
LIN {X 0,Y 121.677,Z 488.793,A -85,B 0,C 180,E1 -27212.619,E2 -27212.619} C_VEL
LIN {X 0,Y 122.254,Z 494.108,A -85,B 0,C 180,E1 -27216.408,E2 -27216.408} C_VEL
LIN {X 0,Y 122.157,Z 498.573,A -85,B 0,C 180,E1 -27219.262,E2 -27219.262} C_VEL
LIN {X 0,Y 122.016,Z 499.45,A -85,B 0,C 180,E1 -27219.779,E2 -27219.779} C_VEL
LIN {X 0,Y 120.903,Z 502.182,A -85,B 0,C 180,E1 -27220.979,E2 -27220.979} C_VEL
LIN {X 0,Y 118.843,Z 505.027,A -85,B 0,C 180,E1 -27221.869,E2 -27221.869} C_VEL
LIN {X 0,Y 111.823,Z 512.433,A -85,B 0,C 180,E1 -27223.929,E2 -27223.929} C_VEL
LIN {X 0,Y 110.297,Z 514.164,A -85,B 0,C 180,E1 -27224.715,E2 -27224.715} C_VEL
LIN {X 0,Y 104.393,Z 521.274,A -85,B 0,C 180,E1 -27228.975,E2 -27228.975} C_VEL
LIN {X 0,Y 97.71,Z 528.321,A -85,B 0,C 180,E1 -27234.872,E2 -27234.872} C_VEL
LIN {X 0,Y 92.97,Z 533.005,A -85,B 0,C 180,E1 -27240.57,E2 -27240.57} C_VEL
LIN {X 0,Y 89.14,Z 536.587,A -85,B 0,C 180,E1 -27246.784,E2 -27246.784} C_VEL
LIN {X 0,Y 87.175,Z 538.434,A -85,B 0,C 180,E1 -27251.188,E2 -27251.188} C_VEL
LIN {X 0,Y 84.679,Z 540.802,A -85,B 0,C 180,E1 -27260.446,E2 -27260.446} C_VEL
LIN {X 0,Y 84.125,Z 541.404,A -85,B 0,C 180,E1 -27265.208,E2 -27265.208} C_VEL
LIN {X 0,Y 83.975,Z 541.627,A -85,B 0,C 180,E1 -27270,E2 -27270} C_VEL
LIN {X 0,Y 84.107,Z 541.431,A -85,B 0,C 180,E1 -27274.794,E2 -27274.794} C_VEL
LIN {X 0,Y 84.68,Z 540.845,A -85,B 0,C 180,E1 -27279.555,E2 -27279.555} C_VEL
LIN {X 0,Y 87.17,Z 538.52,A -85,B 0,C 180,E1 -27288.815,E2 -27288.815} C_VEL
LIN {X 0,Y 90.278,Z 535.65,A -85,B 0,C 180,E1 -27295.352,E2 -27295.352} C_VEL
LIN {X 0,Y 94.334,Z 531.757,A -85,B 0,C 180,E1 -27301.434,E2 -27301.434} C_VEL
LIN {X 0,Y 99.478,Z 526.725,A -85,B 0,C 180,E1 -27306.907,E2 -27306.907} C_VEL
LIN {X 0,Y 105.318,Z 520.388,A -85,B 0,C 180,E1 -27311.861,E2 -27311.861} C_VEL
LIN {X 0,Y 111.473,Z 512.761,A -85,B 0,C 180,E1 -27316.211,E2 -27316.211} C_VEL
LIN {X 0,Y 114.912,Z 507.817,A -85,B 0,C 180,E1 -27318.522,E2 -27318.522} C_VEL
LIN {X 0,Y 116.373,Z 502.71,A -85,B 0,C 180,E1 -27321.73,E2 -27321.73} C_VEL
LIN {X 0,Y 116.894,Z 499.124,A -85,B 0,C 180,E1 -27324.112,E2 -27324.112} C_VEL
LIN {X 0,Y 116.743,Z 494.018,A -85,B 0,C 180,E1 -27328.082,E2 -27328.082} C_VEL
LIN {X 0,Y 116.26,Z 490.61,A -85,B 0,C 180,E1 -27331.079,E2 -27331.079} C_VEL
LIN {X 0,Y 114.926,Z 485.594,A -85,B 0,C 180,E1 -27336.533,E2 -27336.533} C_VEL
LIN {X 0,Y 113.584,Z 481.709,A -85,B 0,C 180,E1 -27341.978,E2 -27341.978} C_VEL
LIN {X 0,Y 112.844,Z 479.697,A -85,B 0,C 180,E1 -27345.574,E2 -27345.574} C_VEL
LIN {X 0,Y 112.298,Z 478.066,A -85,B 0,C 180,E1 -27349.178,E2 -27349.178} C_VEL
LIN {X 0,Y 111.903,Z 475.635,A -85,B 0,C 180,E1 -27360,E2 -27360} C_VEL
LIN {X 0,Y 112.741,Z 478.437,A -85,B 0,C 180,E1 -27370.778,E2 -27370.778} C_VEL
LIN {X 0,Y 113.617,Z 481.329,A -85,B 0,C 180,E1 -27375.845,E2 -27375.845} C_VEL
LIN {X 0,Y 114.07,Z 482.836,A -85,B 0,C 180,E1 -27377.942,E2 -27377.942} C_VEL
LIN {X 0,Y 114.884,Z 487.095,A -85,B 0,C 180,E1 -27382.595,E2 -27382.595} C_VEL
LIN {X 0,Y 115.639,Z 492.039,A -85,B 0,C 180,E1 -27387.117,E2 -27387.117} C_VEL
LIN {X 0,Y 116.079,Z 498.376,A -85,B 0,C 180,E1 -27392.045,E2 -27392.045} C_VEL
LIN {X 0,Y 116.068,Z 502.403,A -85,B 0,C 180,E1 -27394.908,E2 -27394.908} C_VEL
LIN {X 0,Y 114.849,Z 506.724,A -85,B 0,C 180,E1 -27397.296,E2 -27397.296} C_VEL
LIN {X 0,Y 111.313,Z 515.291,A -85,B 0,C 180,E1 -27402.109,E2 -27402.109} C_VEL
LIN {X 0,Y 109.37,Z 518.283,A -85,B 0,C 180,E1 -27403.704,E2 -27403.704} C_VEL
LIN {X 0,Y 102.611,Z 526.407,A -85,B 0,C 180,E1 -27408.629,E2 -27408.629} C_VEL
LIN {X 0,Y 96.514,Z 533.043,A -85,B 0,C 180,E1 -27414.369,E2 -27414.369} C_VEL
LIN {X 0,Y 91.77,Z 537.755,A -85,B 0,C 180,E1 -27420.146,E2 -27420.146} C_VEL
LIN {X 0,Y 88.008,Z 541.358,A -85,B 0,C 180,E1 -27426.466,E2 -27426.466} C_VEL
LIN {X 0,Y 86.238,Z 543.22,A -85,B 0,C 180,E1 -27430.974,E2 -27430.974} C_VEL
LIN {X 0,Y 84.952,Z 544.62,A -85,B 0,C 180,E1 -27435.629,E2 -27435.629} C_VEL
LIN {X 0,Y 84.133,Z 545.621,A -85,B 0,C 180,E1 -27440.382,E2 -27440.382} C_VEL
LIN {X 0,Y 83.787,Z 546.235,A -85,B 0,C 180,E1 -27445.188,E2 -27445.188} C_VEL
LIN {X 0,Y 83.879,Z 546.452,A -85,B 0,C 180,E1 -27450,E2 -27450} C_VEL
LIN {X 0,Y 83.787,Z 546.217,A -85,B 0,C 180,E1 -27454.811,E2 -27454.811} C_VEL
LIN {X 0,Y 84.132,Z 545.593,A -85,B 0,C 180,E1 -27459.617,E2 -27459.617} C_VEL
LIN {X 0,Y 84.951,Z 544.58,A -85,B 0,C 180,E1 -27464.37,E2 -27464.37} C_VEL
LIN {X 0,Y 86.237,Z 543.163,A -85,B 0,C 180,E1 -27469.025,E2 -27469.025} C_VEL
LIN {X 0,Y 89.137,Z 540.203,A -85,B 0,C 180,E1 -27475.699,E2 -27475.699} C_VEL
LIN {X 0,Y 93.232,Z 536.21,A -85,B 0,C 180,E1 -27481.848,E2 -27481.848} C_VEL
LIN {X 0,Y 99.205,Z 530.075,A -85,B 0,C 180,E1 -27488.307,E2 -27488.307} C_VEL
LIN {X 0,Y 105.032,Z 523.376,A -85,B 0,C 180,E1 -27493.303,E2 -27493.303} C_VEL
LIN {X 0,Y 110.416,Z 516.563,A -85,B 0,C 180,E1 -27497.052,E2 -27497.052} C_VEL
LIN {X 0,Y 113.121,Z 510.781,A -85,B 0,C 180,E1 -27500.394,E2 -27500.394} C_VEL
LIN {X 0,Y 115.773,Z 503.424,A -85,B 0,C 180,E1 -27504.302,E2 -27504.302} C_VEL
LIN {X 0,Y 116.008,Z 499.473,A -85,B 0,C 180,E1 -27506.959,E2 -27506.959} C_VEL
LIN {X 0,Y 115.663,Z 492.966,A -85,B 0,C 180,E1 -27511.907,E2 -27511.907} C_VEL
LIN {X 0,Y 114.915,Z 487.708,A -85,B 0,C 180,E1 -27516.545,E2 -27516.545} C_VEL
LIN {X 0,Y 114.598,Z 485.757,A -85,B 0,C 180,E1 -27518.41,E2 -27518.41} C_VEL
LIN {X 0,Y 113.593,Z 481.502,A -85,B 0,C 180,E1 -27523.505,E2 -27523.505} C_VEL
LIN {X 0,Y 112.551,Z 478.219,A -85,B 0,C 180,E1 -27529.203,E2 -27529.203} C_VEL
LIN {X 0,Y 111.799,Z 475.177,A -85,B 0,C 180,E1 -27540,E2 -27540} C_VEL
LIN {X 0,Y 112.085,Z 477.831,A -85,B 0,C 180,E1 -27550.843,E2 -27550.843} C_VEL
LIN {X 0,Y 112.716,Z 479.299,A -85,B 0,C 180,E1 -27554.443,E2 -27554.443} C_VEL
LIN {X 0,Y 113.806,Z 482.601,A -85,B 0,C 180,E1 -27559.856,E2 -27559.856} C_VEL
LIN {X 0,Y 114.633,Z 485.043,A -85,B 0,C 180,E1 -27563.129,E2 -27563.129} C_VEL
LIN {X 0,Y 116.135,Z 490.3,A -85,B 0,C 180,E1 -27568.956,E2 -27568.956} C_VEL
LIN {X 0,Y 116.713,Z 494.755,A -85,B 0,C 180,E1 -27572.816,E2 -27572.816} C_VEL
LIN {X 0,Y 116.654,Z 500.416,A -85,B 0,C 180,E1 -27577.047,E2 -27577.047} C_VEL
LIN {X 0,Y 115.419,Z 505.803,A -85,B 0,C 180,E1 -27580.436,E2 -27580.436} C_VEL
LIN {X 0,Y 114.878,Z 507.458,A -85,B 0,C 180,E1 -27581.459,E2 -27581.459} C_VEL
LIN {X 0,Y 114.064,Z 509.063,A -85,B 0,C 180,E1 -27582.322,E2 -27582.322} C_VEL
LIN {X 0,Y 110.297,Z 514.164,A -85,B 0,C 180,E1 -27584.715,E2 -27584.715} C_VEL
LIN {X 0,Y 106.895,Z 517.787,A -85,B 0,C 180,E1 -27586.457,E2 -27586.457} C_VEL
LIN {X 0,Y 99.982,Z 523.228,A -85,B 0,C 180,E1 -27589,E2 -27589} C_VEL
LIN {X 0,Y 93.044,Z 528.035,A -85,B 0,C 180,E1 -27592.081,E2 -27592.081} C_VEL
LIN {X 0,Y 89.734,Z 530.593,A -85,B 0,C 180,E1 -27594.688,E2 -27594.688} C_VEL
LIN {X 0,Y 83.943,Z 535.734,A -85,B 0,C 180,E1 -27602.582,E2 -27602.582} C_VEL
LIN {X 0,Y 80.472,Z 538.639,A -85,B 0,C 180,E1 -27609.554,E2 -27609.554} C_VEL
LIN {X 0,Y 77.699,Z 541.006,A -85,B 0,C 180,E1 -27619.578,E2 -27619.578} C_VEL
LIN {X 0,Y 77.067,Z 541.608,A -85,B 0,C 180,E1 -27624.768,E2 -27624.768} C_VEL
LIN {X 0,Y 76.896,Z 541.831,A -85,B 0,C 180,E1 -27630.001,E2 -27630.001} C_VEL
LIN {X 0,Y 77.056,Z 541.635,A -85,B 0,C 180,E1 -27635.234,E2 -27635.234} C_VEL
LIN {X 0,Y 77.699,Z 541.049,A -85,B 0,C 180,E1 -27640.423,E2 -27640.423} C_VEL
LIN {X 0,Y 80.465,Z 538.724,A -85,B 0,C 180,E1 -27650.449,E2 -27650.449} C_VEL
LIN {X 0,Y 83.915,Z 535.853,A -85,B 0,C 180,E1 -27657.429,E2 -27657.429} C_VEL
LIN {X 0,Y 88.341,Z 531.96,A -85,B 0,C 180,E1 -27663.841,E2 -27663.841} C_VEL
LIN {X 0,Y 93.889,Z 526.928,A -85,B 0,C 180,E1 -27669.514,E2 -27669.514} C_VEL
LIN {X 0,Y 100.131,Z 520.59,A -85,B 0,C 180,E1 -27674.579,E2 -27674.579} C_VEL
LIN {X 0,Y 106.915,Z 512.67,A -85,B 0,C 180,E1 -27679.106,E2 -27679.106} C_VEL
LIN {X 0,Y 109.214,Z 509.635,A -85,B 0,C 180,E1 -27680.554,E2 -27680.554} C_VEL
LIN {X 0,Y 110.862,Z 504.81,A -85,B 0,C 180,E1 -27683.818,E2 -27683.818} C_VEL
LIN {X 0,Y 111.413,Z 501.559,A -85,B 0,C 180,E1 -27686.29,E2 -27686.29} C_VEL
LIN {X 0,Y 111.46,Z 497.666,A -85,B 0,C 180,E1 -27689.706,E2 -27689.706} C_VEL
LIN {X 0,Y 111.016,Z 493.801,A -85,B 0,C 180,E1 -27693.695,E2 -27693.695} C_VEL
LIN {X 0,Y 110.357,Z 490.71,A -85,B 0,C 180,E1 -27697.536,E2 -27697.536} C_VEL
LIN {X 0,Y 109.364,Z 487.071,A -85,B 0,C 180,E1 -27703.191,E2 -27703.191} C_VEL
LIN {X 0,Y 108.651,Z 484.418,A -85,B 0,C 180,E1 -27708.81,E2 -27708.81} C_VEL
LIN {X 0,Y 108.187,Z 482.585,A -85,B 0,C 180,E1 -27716.275,E2 -27716.275} C_VEL
LIN {X 0,Y 108.48,Z 481.923,A -85,B 0,C 180,E1 -27720,E2 -27720} C_VEL
LIN {X 0,Y 108.593,Z 483.631,A -85,B 0,C 180,E1 -27727.437,E2 -27727.437} C_VEL
LIN {X 0,Y 109.102,Z 484.857,A -85,B 0,C 180,E1 -27731.142,E2 -27731.142} C_VEL
LIN {X 0,Y 109.787,Z 487.745,A -85,B 0,C 180,E1 -27736.213,E2 -27736.213} C_VEL
LIN {X 0,Y 110.278,Z 491.122,A -85,B 0,C 180,E1 -27740.519,E2 -27740.519} C_VEL
LIN {X 0,Y 110.614,Z 495.123,A -85,B 0,C 180,E1 -27744.638,E2 -27744.638} C_VEL
LIN {X 0,Y 110.718,Z 500.606,A -85,B 0,C 180,E1 -27749.467,E2 -27749.467} C_VEL
LIN {X 0,Y 110.468,Z 505.177,A -85,B 0,C 180,E1 -27753.105,E2 -27753.105} C_VEL
LIN {X 0,Y 109.724,Z 507.714,A -85,B 0,C 180,E1 -27754.713,E2 -27754.713} C_VEL
LIN {X 0,Y 106.356,Z 515.074,A -85,B 0,C 180,E1 -27759.064,E2 -27759.064} C_VEL
LIN {X 0,Y 104.56,Z 518.08,A -85,B 0,C 180,E1 -27760.872,E2 -27760.872} C_VEL
LIN {X 0,Y 97.695,Z 525.866,A -85,B 0,C 180,E1 -27765.604,E2 -27765.604} C_VEL
LIN {X 0,Y 90.828,Z 532.84,A -85,B 0,C 180,E1 -27771.755,E2 -27771.755} C_VEL
LIN {X 0,Y 85.663,Z 537.551,A -85,B 0,C 180,E1 -27777.772,E2 -27777.772} C_VEL
LIN {X 0,Y 81.514,Z 541.153,A -85,B 0,C 180,E1 -27784.462,E2 -27784.462} C_VEL
LIN {X 0,Y 79.521,Z 543.016,A -85,B 0,C 180,E1 -27789.297,E2 -27789.297} C_VEL
LIN {X 0,Y 78.057,Z 544.415,A -85,B 0,C 180,E1 -27794.328,E2 -27794.328} C_VEL
LIN {X 0,Y 77.121,Z 545.417,A -85,B 0,C 180,E1 -27799.498,E2 -27799.498} C_VEL
LIN {X 0,Y 76.707,Z 546.031,A -85,B 0,C 180,E1 -27804.743,E2 -27804.743} C_VEL
LIN {X 0,Y 76.777,Z 546.248,A -85,B 0,C 180,E1 -27809.999,E2 -27809.999} C_VEL
LIN {X 0,Y 76.707,Z 546.013,A -85,B 0,C 180,E1 -27815.256,E2 -27815.256} C_VEL
LIN {X 0,Y 77.12,Z 545.388,A -85,B 0,C 180,E1 -27820.501,E2 -27820.501} C_VEL
LIN {X 0,Y 78.056,Z 544.375,A -85,B 0,C 180,E1 -27825.67,E2 -27825.67} C_VEL
LIN {X 0,Y 79.521,Z 542.957,A -85,B 0,C 180,E1 -27830.702,E2 -27830.702} C_VEL
LIN {X 0,Y 82.773,Z 539.997,A -85,B 0,C 180,E1 -27837.838,E2 -27837.838} C_VEL
LIN {X 0,Y 87.243,Z 536.003,A -85,B 0,C 180,E1 -27844.325,E2 -27844.325} C_VEL
LIN {X 0,Y 93.703,Z 529.868,A -85,B 0,C 180,E1 -27851.016,E2 -27851.016} C_VEL
LIN {X 0,Y 99.972,Z 523.17,A -85,B 0,C 180,E1 -27856.101,E2 -27856.101} C_VEL
LIN {X 0,Y 104.531,Z 517.849,A -85,B 0,C 180,E1 -27859.146,E2 -27859.146} C_VEL
LIN {X 0,Y 106.312,Z 514.837,A -85,B 0,C 180,E1 -27860.965,E2 -27860.965} C_VEL
LIN {X 0,Y 109.689,Z 507.445,A -85,B 0,C 180,E1 -27865.297,E2 -27865.297} C_VEL
LIN {X 0,Y 110.394,Z 504.863,A -85,B 0,C 180,E1 -27866.948,E2 -27866.948} C_VEL
LIN {X 0,Y 110.606,Z 500.41,A -85,B 0,C 180,E1 -27870.5,E2 -27870.5} C_VEL
LIN {X 0,Y 110.477,Z 494.69,A -85,B 0,C 180,E1 -27875.543,E2 -27875.543} C_VEL
LIN {X 0,Y 110.137,Z 490.901,A -85,B 0,C 180,E1 -27879.454,E2 -27879.454} C_VEL
LIN {X 0,Y 109.585,Z 487.244,A -85,B 0,C 180,E1 -27884.152,E2 -27884.152} C_VEL
LIN {X 0,Y 108.927,Z 484.636,A -85,B 0,C 180,E1 -27888.84,E2 -27888.84} C_VEL
LIN {X 0,Y 108.189,Z 482.447,A -85,B 0,C 180,E1 -27896.276,E2 -27896.276} C_VEL
LIN {X 0,Y 108.402,Z 481.48,A -85,B 0,C 180,E1 -27900,E2 -27900} C_VEL
LIN {X 0,Y 108.474,Z 484.148,A -85,B 0,C 180,E1 -27911.208,E2 -27911.208} C_VEL
LIN {X 0,Y 108.958,Z 485.78,A -85,B 0,C 180,E1 -27914.952,E2 -27914.952} C_VEL
LIN {X 0,Y 109.815,Z 489.139,A -85,B 0,C 180,E1 -27920.609,E2 -27920.609} C_VEL
LIN {X 0,Y 110.882,Z 493.506,A -85,B 0,C 180,E1 -27926.339,E2 -27926.339} C_VEL
LIN {X 0,Y 111.351,Z 497.361,A -85,B 0,C 180,E1 -27930.327,E2 -27930.327} C_VEL
LIN {X 0,Y 111.289,Z 501.225,A -85,B 0,C 180,E1 -27933.686,E2 -27933.686} C_VEL
LIN {X 0,Y 110.796,Z 504.576,A -85,B 0,C 180,E1 -27936.27,E2 -27936.27} C_VEL
LIN {X 0,Y 109.227,Z 509.278,A -85,B 0,C 180,E1 -27939.456,E2 -27939.456} C_VEL
LIN {X 0,Y 105.547,Z 514.221,A -85,B 0,C 180,E1 -27941.893,E2 -27941.893} C_VEL
LIN {X 0,Y 99.146,Z 521.479,A -85,B 0,C 180,E1 -27946.28,E2 -27946.28} C_VEL
LIN {X 0,Y 92.007,Z 528.526,A -85,B 0,C 180,E1 -27952.333,E2 -27952.333} C_VEL
LIN {X 0,Y 89.734,Z 530.593,A -85,B 0,C 180,E1 -27954.688,E2 -27954.688} C_VEL
LIN {X 0,Y 86.563,Z 532.948,A -85,B 0,C 180,E1 -27957.562,E2 -27957.562} C_VEL
LIN {X 0,Y 80.212,Z 536.249,A -85,B 0,C 180,E1 -27962.294,E2 -27962.294} C_VEL
LIN {X 0,Y 75.407,Z 538.381,A -85,B 0,C 180,E1 -27966.69,E2 -27966.69} C_VEL
LIN {X 0,Y 72.797,Z 539.671,A -85,B 0,C 180,E1 -27970.668,E2 -27970.668} C_VEL
LIN {X 0,Y 72.25,Z 540.013,A -85,B 0,C 180,E1 -27972.13,E2 -27972.13} C_VEL
LIN {X 0,Y 70.717,Z 541.211,A -85,B 0,C 180,E1 -27978.536,E2 -27978.536} C_VEL
LIN {X 0,Y 70.008,Z 541.812,A -85,B 0,C 180,E1 -27984.239,E2 -27984.239} C_VEL
LIN {X 0,Y 69.815,Z 542.034,A -85,B 0,C 180,E1 -27990.001,E2 -27990.001} C_VEL
LIN {X 0,Y 70,Z 541.838,A -85,B 0,C 180,E1 -27995.763,E2 -27995.763} C_VEL
LIN {X 0,Y 72.005,Z 540.286,A -85,B 0,C 180,E1 -28007.027,E2 -28007.027} C_VEL
LIN {X 0,Y 73.848,Z 538.928,A -85,B 0,C 180,E1 -28012.376,E2 -28012.376} C_VEL
LIN {X 0,Y 77.667,Z 536.057,A -85,B 0,C 180,E1 -28019.848,E2 -28019.848} C_VEL
LIN {X 0,Y 82.528,Z 532.163,A -85,B 0,C 180,E1 -28026.593,E2 -28026.593} C_VEL
LIN {X 0,Y 88.525,Z 527.131,A -85,B 0,C 180,E1 -28032.441,E2 -28032.441} C_VEL
LIN {X 0,Y 95.191,Z 520.793,A -85,B 0,C 180,E1 -28037.588,E2 -28037.588} C_VEL
LIN {X 0,Y 102.397,Z 512.872,A -85,B 0,C 180,E1 -28042.117,E2 -28042.117} C_VEL
LIN {X 0,Y 103.626,Z 511.393,A -85,B 0,C 180,E1 -28042.833,E2 -28042.833} C_VEL
LIN {X 0,Y 105.269,Z 507.536,A -85,B 0,C 180,E1 -28045.649,E2 -28045.649} C_VEL
LIN {X 0,Y 105.878,Z 504.835,A -85,B 0,C 180,E1 -28047.925,E2 -28047.925} C_VEL
LIN {X 0,Y 106.145,Z 501.948,A -85,B 0,C 180,E1 -28050.717,E2 -28050.717} C_VEL
LIN {X 0,Y 106.036,Z 498.633,A -85,B 0,C 180,E1 -28054.48,E2 -28054.48} C_VEL
LIN {X 0,Y 105.586,Z 495.553,A -85,B 0,C 180,E1 -28058.73,E2 -28058.73} C_VEL
LIN {X 0,Y 104.951,Z 492.265,A -85,B 0,C 180,E1 -28064.463,E2 -28064.463} C_VEL
LIN {X 0,Y 104.647,Z 490.585,A -85,B 0,C 180,E1 -28068.376,E2 -28068.376} C_VEL
LIN {X 0,Y 104.39,Z 489.405,A -85,B 0,C 180,E1 -28072.261,E2 -28072.261} C_VEL
LIN {X 0,Y 104.681,Z 487.977,A -85,B 0,C 180,E1 -28080,E2 -28080} C_VEL
LIN {X 0,Y 104.717,Z 489.712,A -85,B 0,C 180,E1 -28087.714,E2 -28087.714} C_VEL
LIN {X 0,Y 105.127,Z 491.055,A -85,B 0,C 180,E1 -28091.569,E2 -28091.569} C_VEL
LIN {X 0,Y 105.429,Z 493.188,A -85,B 0,C 180,E1 -28095.464,E2 -28095.464} C_VEL
LIN {X 0,Y 105.615,Z 496.077,A -85,B 0,C 180,E1 -28099.434,E2 -28099.434} C_VEL
LIN {X 0,Y 105.588,Z 500.767,A -85,B 0,C 180,E1 -28104.582,E2 -28104.582} C_VEL
LIN {X 0,Y 105.173,Z 506.228,A -85,B 0,C 180,E1 -28109.691,E2 -28109.691} C_VEL
LIN {X 0,Y 104.701,Z 508.869,A -85,B 0,C 180,E1 -28111.933,E2 -28111.933} C_VEL
LIN {X 0,Y 100.824,Z 516.368,A -85,B 0,C 180,E1 -28116.715,E2 -28116.715} C_VEL
LIN {X 0,Y 99.938,Z 517.872,A -85,B 0,C 180,E1 -28117.707,E2 -28117.707} C_VEL
LIN {X 0,Y 92.831,Z 525.551,A -85,B 0,C 180,E1 -28122.427,E2 -28122.427} C_VEL
LIN {X 0,Y 85.353,Z 532.637,A -85,B 0,C 180,E1 -28128.797,E2 -28128.797} C_VEL
LIN {X 0,Y 79.726,Z 537.348,A -85,B 0,C 180,E1 -28135.04,E2 -28135.04} C_VEL
LIN {X 0,Y 75.14,Z 540.949,A -85,B 0,C 180,E1 -28142.117,E2 -28142.117} C_VEL
LIN {X 0,Y 72.893,Z 542.812,A -85,B 0,C 180,E1 -28147.315,E2 -28147.315} C_VEL
LIN {X 0,Y 70.142,Z 545.213,A -85,B 0,C 180,E1 -28158.439,E2 -28158.439} C_VEL
LIN {X 0,Y 69.621,Z 545.826,A -85,B 0,C 180,E1 -28164.206,E2 -28164.206} C_VEL
LIN {X 0,Y 69.698,Z 546.044,A -85,B 0,C 180,E1 -28169.999,E2 -28169.999} C_VEL
LIN {X 0,Y 69.621,Z 545.808,A -85,B 0,C 180,E1 -28175.793,E2 -28175.793} C_VEL
LIN {X 0,Y 70.142,Z 545.183,A -85,B 0,C 180,E1 -28181.559,E2 -28181.559} C_VEL
LIN {X 0,Y 71.219,Z 544.169,A -85,B 0,C 180,E1 -28187.22,E2 -28187.22} C_VEL
LIN {X 0,Y 72.893,Z 542.752,A -85,B 0,C 180,E1 -28192.684,E2 -28192.684} C_VEL
LIN {X 0,Y 76.548,Z 539.792,A -85,B 0,C 180,E1 -28200.329,E2 -28200.329} C_VEL
LIN {X 0,Y 81.445,Z 535.797,A -85,B 0,C 180,E1 -28207.159,E2 -28207.159} C_VEL
LIN {X 0,Y 87.4,Z 530.666,A -85,B 0,C 180,E1 -28213.117,E2 -28213.117} C_VEL
LIN {X 0,Y 95.158,Z 522.963,A -85,B 0,C 180,E1 -28219.202,E2 -28219.202} C_VEL
LIN {X 0,Y 99.905,Z 517.636,A -85,B 0,C 180,E1 -28222.316,E2 -28222.316} C_VEL
LIN {X 0,Y 104.167,Z 509.784,A -85,B 0,C 180,E1 -28227.333,E2 -28227.333} C_VEL
LIN {X 0,Y 104.872,Z 507.536,A -85,B 0,C 180,E1 -28228.951,E2 -28228.951} C_VEL
LIN {X 0,Y 105.455,Z 501.63,A -85,B 0,C 180,E1 -28234.33,E2 -28234.33} C_VEL
LIN {X 0,Y 105.513,Z 497.343,A -85,B 0,C 180,E1 -28238.829,E2 -28238.829} C_VEL
LIN {X 0,Y 105.312,Z 493.684,A -85,B 0,C 180,E1 -28243.491,E2 -28243.491} C_VEL
LIN {X 0,Y 105.116,Z 491.858,A -85,B 0,C 180,E1 -28246.467,E2 -28246.467} C_VEL
LIN {X 0,Y 104.939,Z 490.873,A -85,B 0,C 180,E1 -28248.41,E2 -28248.41} C_VEL
